LIN {X 0,Y 468.143,Z 375.937,A -85,B 0,C 180,E1 -7618.838,E2 -7618.838} C_VEL
LIN {X 0,Y 467.826,Z 382.891,A -85,B 0,C 180,E1 -7621.757,E2 -7621.757} C_VEL
LIN {X 0,Y 467.602,Z 389.263,A -85,B 0,C 180,E1 -7624.395,E2 -7624.395} C_VEL
LIN {X 0,Y 467.33,Z 397.834,A -85,B 0,C 180,E1 -7627.916,E2 -7627.916} C_VEL
LIN {X 0,Y 467.292,Z 398.559,A -85,B 0,C 180,E1 -7628.21,E2 -7628.21} C_VEL
LIN {X 0,Y 471.188,Z 415.228,A -85,B 0,C 180,E1 -7628.746,E2 -7628.746} C_VEL
LIN {X 0,Y 473.512,Z 427.366,A -85,B 0,C 180,E1 -7629.238,E2 -7629.238} C_VEL
LIN {X 0,Y 472.916,Z 441.368,A -85,B 0,C 180,E1 -7629.804,E2 -7629.804} C_VEL
LIN {X 0,Y 472.102,Z 455.526,A -85,B 0,C 180,E1 -7630.544,E2 -7630.544} C_VEL
LIN {X 0,Y 471.29,Z 468.776,A -85,B 0,C 180,E1 -7631.413,E2 -7631.413} C_VEL
LIN {X 0,Y 470.385,Z 482.274,A -85,B 0,C 180,E1 -7632.502,E2 -7632.502} C_VEL
LIN {X 0,Y 469.612,Z 494.581,A -85,B 0,C 180,E1 -7633.704,E2 -7633.704} C_VEL
LIN {X 0,Y 468.781,Z 505.819,A -85,B 0,C 180,E1 -7635.013,E2 -7635.013} C_VEL
LIN {X 0,Y 468.067,Z 516.736,A -85,B 0,C 180,E1 -7636.542,E2 -7636.542} C_VEL
LIN {X 0,Y 467.596,Z 525.839,A -85,B 0,C 180,E1 -7638.073,E2 -7638.073} C_VEL
LIN {X 0,Y 467.244,Z 533.393,A -85,B 0,C 180,E1 -7639.602,E2 -7639.602} C_VEL
LIN {X 0,Y 466.93,Z 540.444,A -85,B 0,C 180,E1 -7641.344,E2 -7641.344} C_VEL
LIN {X 0,Y 466.818,Z 545.996,A -85,B 0,C 180,E1 -7643.083,E2 -7643.083} C_VEL
LIN {X 0,Y 466.694,Z 550.191,A -85,B 0,C 180,E1 -7644.816,E2 -7644.816} C_VEL
LIN {X 0,Y 466.705,Z 553.137,A -85,B 0,C 180,E1 -7646.547,E2 -7646.547} C_VEL
LIN {X 0,Y 466.652,Z 554.892,A -85,B 0,C 180,E1 -7648.274,E2 -7648.274} C_VEL
LIN {X 0,Y 466.595,Z 555.491,A -85,B 0,C 180,E1 -7650,E2 -7650} C_VEL
LIN {X 0,Y 466.652,Z 554.889,A -85,B 0,C 180,E1 -7651.726,E2 -7651.726} C_VEL
LIN {X 0,Y 466.705,Z 553.132,A -85,B 0,C 180,E1 -7653.454,E2 -7653.454} C_VEL
LIN {X 0,Y 466.721,Z 550.189,A -85,B 0,C 180,E1 -7655.184,E2 -7655.184} C_VEL
LIN {X 0,Y 466.822,Z 545.998,A -85,B 0,C 180,E1 -7656.918,E2 -7656.918} C_VEL
LIN {X 0,Y 466.93,Z 540.443,A -85,B 0,C 180,E1 -7658.657,E2 -7658.657} C_VEL
LIN {X 0,Y 467.245,Z 533.383,A -85,B 0,C 180,E1 -7660.399,E2 -7660.399} C_VEL
LIN {X 0,Y 467.612,Z 525.832,A -85,B 0,C 180,E1 -7661.927,E2 -7661.927} C_VEL
LIN {X 0,Y 468.068,Z 516.733,A -85,B 0,C 180,E1 -7663.458,E2 -7663.458} C_VEL
LIN {X 0,Y 468.76,Z 505.812,A -85,B 0,C 180,E1 -7664.989,E2 -7664.989} C_VEL
LIN {X 0,Y 469.61,Z 493.547,A -85,B 0,C 180,E1 -7666.408,E2 -7666.408} C_VEL
LIN {X 0,Y 470.458,Z 481.048,A -85,B 0,C 180,E1 -7667.609,E2 -7667.609} C_VEL
LIN {X 0,Y 471.366,Z 467.232,A -85,B 0,C 180,E1 -7668.697,E2 -7668.697} C_VEL
LIN {X 0,Y 472.233,Z 453.677,A -85,B 0,C 180,E1 -7669.564,E2 -7669.564} C_VEL
LIN {X 0,Y 472.939,Z 439.651,A -85,B 0,C 180,E1 -7670.28,E2 -7670.28} C_VEL
LIN {X 0,Y 473.403,Z 425.835,A -85,B 0,C 180,E1 -7670.823,E2 -7670.823} C_VEL
LIN {X 0,Y 470.06,Z 410.115,A -85,B 0,C 180,E1 -7671.434,E2 -7671.434} C_VEL
LIN {X 0,Y 467.287,Z 398.544,A -85,B 0,C 180,E1 -7671.794,E2 -7671.794} C_VEL
LIN {X 0,Y 467.513,Z 390.984,A -85,B 0,C 180,E1 -7674.893,E2 -7674.893} C_VEL
LIN {X 0,Y 467.773,Z 384.017,A -85,B 0,C 180,E1 -7677.759,E2 -7677.759} C_VEL
LIN {X 0,Y 468.035,Z 376.994,A -85,B 0,C 180,E1 -7680.7,E2 -7680.7} C_VEL
LIN {X 0,Y 468.345,Z 369.941,A -85,B 0,C 180,E1 -7683.726,E2 -7683.726} C_VEL
LIN {X 0,Y 468.684,Z 364.077,A -85,B 0,C 180,E1 -7686.34,E2 -7686.34} C_VEL
LIN {X 0,Y 468.997,Z 357.229,A -85,B 0,C 180,E1 -7689.559,E2 -7689.559} C_VEL
LIN {X 0,Y 469.127,Z 353.286,A -85,B 0,C 180,E1 -7691.492,E2 -7691.492} C_VEL
LIN {X 0,Y 468.587,Z 348.664,A -85,B 0,C 180,E1 -7693.952,E2 -7693.952} C_VEL
LIN {X 0,Y 467.687,Z 343.617,A -85,B 0,C 180,E1 -7696.865,E2 -7696.865} C_VEL
LIN {X 0,Y 467.591,Z 342.867,A -85,B 0,C 180,E1 -7697.44,E2 -7697.44} C_VEL
LIN {X 0,Y 467.584,Z 342.869,A -85,B 0,C 180,E1 -7700.856,E2 -7700.856} C_VEL
LIN {X 0,Y 467.566,Z 342.872,A -85,B 0,C 180,E1 -7704.261,E2 -7704.261} C_VEL
LIN {X 0,Y 467.584,Z 342.868,A -85,B 0,C 180,E1 -7707.321,E2 -7707.321} C_VEL
LIN {X 0,Y 467.573,Z 342.87,A -85,B 0,C 180,E1 -7710.668,E2 -7710.668} C_VEL
LIN {X 0,Y 467.618,Z 342.862,A -85,B 0,C 180,E1 -7713.2,E2 -7713.2} C_VEL
LIN {X 0,Y 467.595,Z 342.864,A -85,B 0,C 180,E1 -7716.468,E2 -7716.468} C_VEL
LIN {X 0,Y 467.626,Z 342.863,A -85,B 0,C 180,E1 -7719.777,E2 -7719.777} C_VEL
LIN {X 0,Y 467.612,Z 342.862,A -85,B 0,C 180,E1 -7722.507,E2 -7722.507} C_VEL
LIN {X 0,Y 467.61,Z 342.864,A -85,B 0,C 180,E1 -7725.197,E2 -7725.197} C_VEL
LIN {X 0,Y 467.659,Z 342.86,A -85,B 0,C 180,E1 -7727.855,E2 -7727.855} C_VEL
LIN {X 0,Y 467.685,Z 342.853,A -85,B 0,C 180,E1 -7731.357,E2 -7731.357} C_VEL
LIN {X 0,Y 467.747,Z 342.847,A -85,B 0,C 180,E1 -7733.963,E2 -7733.963} C_VEL
LIN {X 0,Y 467.863,Z 342.83,A -85,B 0,C 180,E1 -7737.417,E2 -7737.417} C_VEL
LIN {X 0,Y 467.885,Z 342.829,A -85,B 0,C 180,E1 -7740,E2 -7740} C_VEL
LIN {X 0,Y 467.863,Z 342.832,A -85,B 0,C 180,E1 -7742.583,E2 -7742.583} C_VEL
LIN {X 0,Y 467.748,Z 342.846,A -85,B 0,C 180,E1 -7746.037,E2 -7746.037} C_VEL
LIN {X 0,Y 467.686,Z 342.854,A -85,B 0,C 180,E1 -7748.643,E2 -7748.643} C_VEL
LIN {X 0,Y 467.659,Z 342.844,A -85,B 0,C 180,E1 -7752.145,E2 -7752.145} C_VEL
LIN {X 0,Y 467.643,Z 342.856,A -85,B 0,C 180,E1 -7755.695,E2 -7755.695} C_VEL
LIN {X 0,Y 467.621,Z 342.855,A -85,B 0,C 180,E1 -7758.765,E2 -7758.765} C_VEL
LIN {X 0,Y 467.584,Z 342.858,A -85,B 0,C 180,E1 -7761.268,E2 -7761.268} C_VEL
LIN {X 0,Y 467.566,Z 342.869,A -85,B 0,C 180,E1 -7763.944,E2 -7763.944} C_VEL
LIN {X 0,Y 467.616,Z 342.855,A -85,B 0,C 180,E1 -7766.8,E2 -7766.8} C_VEL
LIN {X 0,Y 467.557,Z 342.868,A -85,B 0,C 180,E1 -7769.738,E2 -7769.738} C_VEL
LIN {X 0,Y 467.586,Z 342.86,A -85,B 0,C 180,E1 -7772.758,E2 -7772.758} C_VEL
LIN {X 0,Y 467.559,Z 342.868,A -85,B 0,C 180,E1 -7775.889,E2 -7775.889} C_VEL
LIN {X 0,Y 467.586,Z 342.867,A -85,B 0,C 180,E1 -7779.145,E2 -7779.145} C_VEL
LIN {X 0,Y 467.589,Z 342.869,A -85,B 0,C 180,E1 -7782.567,E2 -7782.567} C_VEL
LIN {X 0,Y 467.573,Z 342.869,A -85,B 0,C 180,E1 -7785.053,E2 -7785.053} C_VEL
LIN {X 0,Y 467.545,Z 342.874,A -85,B 0,C 180,E1 -7787.439,E2 -7787.439} C_VEL
LIN {X 0,Y 467.333,Z 342.9,A -85,B 0,C 180,E1 -7790.082,E2 -7790.082} C_VEL
LIN {X 0,Y 467.23,Z 343.077,A -85,B 0,C 180,E1 -7791.46,E2 -7791.46} C_VEL
LIN {X 0,Y 467.185,Z 345.526,A -85,B 0,C 180,E1 -7794.325,E2 -7794.325} C_VEL
LIN {X 0,Y 467.138,Z 348.226,A -85,B 0,C 180,E1 -7797.406,E2 -7797.406} C_VEL
LIN {X 0,Y 467.036,Z 351.246,A -85,B 0,C 180,E1 -7800.785,E2 -7800.785} C_VEL
LIN {X 0,Y 466.95,Z 354.424,A -85,B 0,C 180,E1 -7804.12,E2 -7804.12} C_VEL
LIN {X 0,Y 466.89,Z 357.26,A -85,B 0,C 180,E1 -7806.96,E2 -7806.96} C_VEL
LIN {X 0,Y 466.856,Z 358.631,A -85,B 0,C 180,E1 -7808.273,E2 -7808.273} C_VEL
LIN {X 0,Y 472.012,Z 374.868,A -85,B 0,C 180,E1 -7808.908,E2 -7808.908} C_VEL
LIN {X 0,Y 473.883,Z 382.02,A -85,B 0,C 180,E1 -7809.228,E2 -7809.228} C_VEL
LIN {X 0,Y 473.379,Z 397.457,A -85,B 0,C 180,E1 -7809.851,E2 -7809.851} C_VEL
LIN {X 0,Y 472.672,Z 411.134,A -85,B 0,C 180,E1 -7810.568,E2 -7810.568} C_VEL
LIN {X 0,Y 472.562,Z 413.419,A -85,B 0,C 180,E1 -7810.71,E2 -7810.71} C_VEL
LIN {X 0,Y 471.674,Z 418.718,A -85,B 0,C 180,E1 -7811.02,E2 -7811.02} C_VEL
LIN {X 0,Y 468.437,Z 427.17,A -85,B 0,C 180,E1 -7811.503,E2 -7811.503} C_VEL
LIN {X 0,Y 465.109,Z 435.383,A -85,B 0,C 180,E1 -7812.047,E2 -7812.047} C_VEL
LIN {X 0,Y 464.087,Z 440.168,A -85,B 0,C 180,E1 -7812.453,E2 -7812.453} C_VEL
LIN {X 0,Y 463.172,Z 452.261,A -85,B 0,C 180,E1 -7813.697,E2 -7813.697} C_VEL
LIN {X 0,Y 462.349,Z 463.033,A -85,B 0,C 180,E1 -7815.024,E2 -7815.024} C_VEL
LIN {X 0,Y 461.661,Z 472.162,A -85,B 0,C 180,E1 -7816.351,E2 -7816.351} C_VEL
LIN {X 0,Y 461.067,Z 481.078,A -85,B 0,C 180,E1 -7817.901,E2 -7817.901} C_VEL
LIN {X 0,Y 460.524,Z 488.466,A -85,B 0,C 180,E1 -7819.447,E2 -7819.447} C_VEL
LIN {X 0,Y 460.187,Z 495.365,A -85,B 0,C 180,E1 -7821.215,E2 -7821.215} C_VEL
LIN {X 0,Y 459.916,Z 500.786,A -85,B 0,C 180,E1 -7822.978,E2 -7822.978} C_VEL
LIN {X 0,Y 459.699,Z 504.881,A -85,B 0,C 180,E1 -7824.737,E2 -7824.737} C_VEL
LIN {X 0,Y 459.689,Z 507.753,A -85,B 0,C 180,E1 -7826.494,E2 -7826.494} C_VEL
LIN {X 0,Y 459.631,Z 509.485,A -85,B 0,C 180,E1 -7828.247,E2 -7828.247} C_VEL
LIN {X 0,Y 459.528,Z 510.096,A -85,B 0,C 180,E1 -7830,E2 -7830} C_VEL
LIN {X 0,Y 459.632,Z 509.536,A -85,B 0,C 180,E1 -7831.752,E2 -7831.752} C_VEL
LIN {X 0,Y 459.689,Z 507.872,A -85,B 0,C 180,E1 -7833.506,E2 -7833.506} C_VEL
LIN {X 0,Y 459.694,Z 505.065,A -85,B 0,C 180,E1 -7835.263,E2 -7835.263} C_VEL
LIN {X 0,Y 459.908,Z 501.035,A -85,B 0,C 180,E1 -7837.022,E2 -7837.022} C_VEL
LIN {X 0,Y 460.182,Z 495.691,A -85,B 0,C 180,E1 -7838.784,E2 -7838.784} C_VEL
LIN {X 0,Y 460.498,Z 488.881,A -85,B 0,C 180,E1 -7840.552,E2 -7840.552} C_VEL
LIN {X 0,Y 461.022,Z 481.546,A -85,B 0,C 180,E1 -7842.099,E2 -7842.099} C_VEL
LIN {X 0,Y 461.624,Z 472.707,A -85,B 0,C 180,E1 -7843.649,E2 -7843.649} C_VEL
LIN {X 0,Y 462.296,Z 463.688,A -85,B 0,C 180,E1 -7844.977,E2 -7844.977} C_VEL
LIN {X 0,Y 463.089,Z 453.042,A -85,B 0,C 180,E1 -7846.305,E2 -7846.305} C_VEL
LIN {X 0,Y 463.997,Z 441.752,A -85,B 0,C 180,E1 -7847.486,E2 -7847.486} C_VEL
LIN {X 0,Y 464.916,Z 428.697,A -85,B 0,C 180,E1 -7848.623,E2 -7848.623} C_VEL
LIN {X 0,Y 465.751,Z 414.664,A -85,B 0,C 180,E1 -7849.617,E2 -7849.617} C_VEL
LIN {X 0,Y 466.589,Z 400.159,A -85,B 0,C 180,E1 -7850.427,E2 -7850.427} C_VEL
LIN {X 0,Y 467.191,Z 384.917,A -85,B 0,C 180,E1 -7851.078,E2 -7851.078} C_VEL
LIN {X 0,Y 467.053,Z 382.296,A -85,B 0,C 180,E1 -7851.184,E2 -7851.184} C_VEL
LIN {X 0,Y 462.919,Z 368.608,A -85,B 0,C 180,E1 -7851.802,E2 -7851.802} C_VEL
LIN {X 0,Y 459.771,Z 358.928,A -85,B 0,C 180,E1 -7852.186,E2 -7852.186} C_VEL
LIN {X 0,Y 459.889,Z 355.488,A -85,B 0,C 180,E1 -7855.626,E2 -7855.626} C_VEL
LIN {X 0,Y 459.941,Z 352.956,A -85,B 0,C 180,E1 -7858.273,E2 -7858.273} C_VEL
LIN {X 0,Y 460.006,Z 350.233,A -85,B 0,C 180,E1 -7861.295,E2 -7861.295} C_VEL
LIN {X 0,Y 460.124,Z 347.516,A -85,B 0,C 180,E1 -7864.431,E2 -7864.431} C_VEL
LIN {X 0,Y 460.157,Z 344.726,A -85,B 0,C 180,E1 -7867.656,E2 -7867.656} C_VEL
LIN {X 0,Y 460.17,Z 343.794,A -85,B 0,C 180,E1 -7868.84,E2 -7868.84} C_VEL
LIN {X 0,Y 460.455,Z 343.754,A -85,B 0,C 180,E1 -7871.591,E2 -7871.591} C_VEL
LIN {X 0,Y 460.515,Z 343.749,A -85,B 0,C 180,E1 -7874.588,E2 -7874.588} C_VEL
LIN {X 0,Y 460.521,Z 343.748,A -85,B 0,C 180,E1 -7877.818,E2 -7877.818} C_VEL
LIN {X 0,Y 460.544,Z 343.742,A -85,B 0,C 180,E1 -7881.102,E2 -7881.102} C_VEL
LIN {X 0,Y 460.513,Z 343.746,A -85,B 0,C 180,E1 -7884.554,E2 -7884.554} C_VEL
LIN {X 0,Y 460.531,Z 343.738,A -85,B 0,C 180,E1 -7887.715,E2 -7887.715} C_VEL
LIN {X 0,Y 460.546,Z 343.741,A -85,B 0,C 180,E1 -7890.769,E2 -7890.769} C_VEL
LIN {X 0,Y 460.567,Z 343.732,A -85,B 0,C 180,E1 -7893.735,E2 -7893.735} C_VEL
LIN {X 0,Y 460.544,Z 343.741,A -85,B 0,C 180,E1 -7896.624,E2 -7896.624} C_VEL
LIN {X 0,Y 460.55,Z 343.729,A -85,B 0,C 180,E1 -7899.453,E2 -7899.453} C_VEL
LIN {X 0,Y 460.558,Z 343.742,A -85,B 0,C 180,E1 -7902.23,E2 -7902.23} C_VEL
LIN {X 0,Y 460.564,Z 343.738,A -85,B 0,C 180,E1 -7904.965,E2 -7904.965} C_VEL
LIN {X 0,Y 460.628,Z 343.721,A -85,B 0,C 180,E1 -7907.666,E2 -7907.666} C_VEL
LIN {X 0,Y 460.627,Z 343.734,A -85,B 0,C 180,E1 -7911.224,E2 -7911.224} C_VEL
LIN {X 0,Y 460.709,Z 343.723,A -85,B 0,C 180,E1 -7913.87,E2 -7913.87} C_VEL
LIN {X 0,Y 460.823,Z 343.71,A -85,B 0,C 180,E1 -7917.378,E2 -7917.378} C_VEL
LIN {X 0,Y 460.851,Z 343.707,A -85,B 0,C 180,E1 -7920,E2 -7920} C_VEL
LIN {X 0,Y 460.824,Z 343.707,A -85,B 0,C 180,E1 -7922.622,E2 -7922.622} C_VEL
LIN {X 0,Y 460.708,Z 343.725,A -85,B 0,C 180,E1 -7926.13,E2 -7926.13} C_VEL
LIN {X 0,Y 460.627,Z 343.732,A -85,B 0,C 180,E1 -7928.776,E2 -7928.776} C_VEL
LIN {X 0,Y 460.611,Z 343.734,A -85,B 0,C 180,E1 -7932.445,E2 -7932.445} C_VEL
LIN {X 0,Y 460.597,Z 343.734,A -85,B 0,C 180,E1 -7935.998,E2 -7935.998} C_VEL
LIN {X 0,Y 460.569,Z 343.74,A -85,B 0,C 180,E1 -7938.902,E2 -7938.902} C_VEL
LIN {X 0,Y 460.514,Z 343.749,A -85,B 0,C 180,E1 -7941.486,E2 -7941.486} C_VEL
LIN {X 0,Y 460.54,Z 343.746,A -85,B 0,C 180,E1 -7944.332,E2 -7944.332} C_VEL
LIN {X 0,Y 460.577,Z 343.741,A -85,B 0,C 180,E1 -7947.243,E2 -7947.243} C_VEL
LIN {X 0,Y 460.525,Z 343.746,A -85,B 0,C 180,E1 -7950.239,E2 -7950.239} C_VEL
LIN {X 0,Y 460.527,Z 343.747,A -85,B 0,C 180,E1 -7953.325,E2 -7953.325} C_VEL
LIN {X 0,Y 460.477,Z 343.753,A -85,B 0,C 180,E1 -7956.529,E2 -7956.529} C_VEL
LIN {X 0,Y 460.556,Z 343.744,A -85,B 0,C 180,E1 -7959.86,E2 -7959.86} C_VEL
LIN {X 0,Y 460.549,Z 343.823,A -85,B 0,C 180,E1 -7962.368,E2 -7962.368} C_VEL
LIN {X 0,Y 461.49,Z 349.212,A -85,B 0,C 180,E1 -7965.531,E2 -7965.531} C_VEL
LIN {X 0,Y 462.108,Z 354.056,A -85,B 0,C 180,E1 -7968.178,E2 -7968.178} C_VEL
LIN {X 0,Y 462.055,Z 358.224,A -85,B 0,C 180,E1 -7970.296,E2 -7970.296} C_VEL
LIN {X 0,Y 461.674,Z 365.567,A -85,B 0,C 180,E1 -7973.785,E2 -7973.785} C_VEL
LIN {X 0,Y 461.28,Z 372.537,A -85,B 0,C 180,E1 -7976.927,E2 -7976.927} C_VEL
LIN {X 0,Y 460.999,Z 379.111,A -85,B 0,C 180,E1 -7979.796,E2 -7979.796} C_VEL
LIN {X 0,Y 460.668,Z 386.088,A -85,B 0,C 180,E1 -7982.763,E2 -7982.763} C_VEL
LIN {X 0,Y 460.411,Z 392.987,A -85,B 0,C 180,E1 -7985.661,E2 -7985.661} C_VEL
LIN {X 0,Y 460.252,Z 398.18,A -85,B 0,C 180,E1 -7987.848,E2 -7987.848} C_VEL
LIN {X 0,Y 464.531,Z 416.477,A -85,B 0,C 180,E1 -7988.469,E2 -7988.469} C_VEL
LIN {X 0,Y 466.803,Z 428.417,A -85,B 0,C 180,E1 -7988.979,E2 -7988.979} C_VEL
LIN {X 0,Y 466.202,Z 441.436,A -85,B 0,C 180,E1 -7989.521,E2 -7989.521} C_VEL
LIN {X 0,Y 465.391,Z 455.18,A -85,B 0,C 180,E1 -7990.252,E2 -7990.252} C_VEL
LIN {X 0,Y 464.469,Z 468.425,A -85,B 0,C 180,E1 -7991.13,E2 -7991.13} C_VEL
LIN {X 0,Y 463.542,Z 481.925,A -85,B 0,C 180,E1 -7992.235,E2 -7992.235} C_VEL
LIN {X 0,Y 462.707,Z 494.23,A -85,B 0,C 180,E1 -7993.454,E2 -7993.454} C_VEL
LIN {X 0,Y 461.839,Z 505.468,A -85,B 0,C 180,E1 -7994.782,E2 -7994.782} C_VEL
LIN {X 0,Y 461.082,Z 516.385,A -85,B 0,C 180,E1 -7996.335,E2 -7996.335} C_VEL
LIN {X 0,Y 460.551,Z 525.486,A -85,B 0,C 180,E1 -7997.888,E2 -7997.888} C_VEL
LIN {X 0,Y 460.194,Z 533.042,A -85,B 0,C 180,E1 -7999.441,E2 -7999.441} C_VEL
LIN {X 0,Y 459.868,Z 540.094,A -85,B 0,C 180,E1 -8001.21,E2 -8001.21} C_VEL
LIN {X 0,Y 459.728,Z 545.646,A -85,B 0,C 180,E1 -8002.976,E2 -8002.976} C_VEL
LIN {X 0,Y 459.605,Z 549.843,A -85,B 0,C 180,E1 -8004.736,E2 -8004.736} C_VEL
LIN {X 0,Y 459.601,Z 552.789,A -85,B 0,C 180,E1 -8006.494,E2 -8006.494} C_VEL
LIN {X 0,Y 459.56,Z 554.544,A -85,B 0,C 180,E1 -8008.248,E2 -8008.248} C_VEL
LIN {X 0,Y 459.527,Z 555.144,A -85,B 0,C 180,E1 -8010,E2 -8010} C_VEL
LIN {X 0,Y 459.56,Z 554.541,A -85,B 0,C 180,E1 -8011.753,E2 -8011.753} C_VEL
LIN {X 0,Y 459.601,Z 552.783,A -85,B 0,C 180,E1 -8013.507,E2 -8013.507} C_VEL
LIN {X 0,Y 459.631,Z 549.84,A -85,B 0,C 180,E1 -8015.264,E2 -8015.264} C_VEL
LIN {X 0,Y 459.73,Z 545.648,A -85,B 0,C 180,E1 -8017.025,E2 -8017.025} C_VEL
LIN {X 0,Y 459.869,Z 540.093,A -85,B 0,C 180,E1 -8018.791,E2 -8018.791} C_VEL
LIN {X 0,Y 460.195,Z 533.032,A -85,B 0,C 180,E1 -8020.56,E2 -8020.56} C_VEL
LIN {X 0,Y 460.562,Z 525.478,A -85,B 0,C 180,E1 -8022.112,E2 -8022.112} C_VEL
LIN {X 0,Y 461.084,Z 516.38,A -85,B 0,C 180,E1 -8023.666,E2 -8023.666} C_VEL
LIN {X 0,Y 461.812,Z 505.458,A -85,B 0,C 180,E1 -8025.22,E2 -8025.22} C_VEL
LIN {X 0,Y 462.717,Z 493.193,A -85,B 0,C 180,E1 -8026.66,E2 -8026.66} C_VEL
LIN {X 0,Y 463.613,Z 480.694,A -85,B 0,C 180,E1 -8027.877,E2 -8027.877} C_VEL
LIN {X 0,Y 464.603,Z 466.879,A -85,B 0,C 180,E1 -8028.98,E2 -8028.98} C_VEL
LIN {X 0,Y 465.519,Z 453.324,A -85,B 0,C 180,E1 -8029.858,E2 -8029.858} C_VEL
LIN {X 0,Y 466.252,Z 438.42,A -85,B 0,C 180,E1 -8030.625,E2 -8030.625} C_VEL
LIN {X 0,Y 466.736,Z 427.317,A -85,B 0,C 180,E1 -8031.066,E2 -8031.066} C_VEL
LIN {X 0,Y 463.453,Z 411.48,A -85,B 0,C 180,E1 -8031.711,E2 -8031.711} C_VEL
LIN {X 0,Y 460.254,Z 398.191,A -85,B 0,C 180,E1 -8032.145,E2 -8032.145} C_VEL
LIN {X 0,Y 460.581,Z 389.454,A -85,B 0,C 180,E1 -8035.805,E2 -8035.805} C_VEL
LIN {X 0,Y 460.894,Z 381.437,A -85,B 0,C 180,E1 -8039.207,E2 -8039.207} C_VEL
LIN {X 0,Y 461.193,Z 374.372,A -85,B 0,C 180,E1 -8042.233,E2 -8042.233} C_VEL
LIN {X 0,Y 461.538,Z 367.371,A -85,B 0,C 180,E1 -8045.355,E2 -8045.355} C_VEL
LIN {X 0,Y 461.776,Z 362.393,A -85,B 0,C 180,E1 -8047.682,E2 -8047.682} C_VEL
LIN {X 0,Y 462.141,Z 355.905,A -85,B 0,C 180,E1 -8050.838,E2 -8050.838} C_VEL
LIN {X 0,Y 461.835,Z 351.65,A -85,B 0,C 180,E1 -8053.077,E2 -8053.077} C_VEL
LIN {X 0,Y 461.091,Z 346.925,A -85,B 0,C 180,E1 -8055.757,E2 -8055.757} C_VEL
LIN {X 0,Y 460.526,Z 343.748,A -85,B 0,C 180,E1 -8057.724,E2 -8057.724} C_VEL
LIN {X 0,Y 460.547,Z 343.746,A -85,B 0,C 180,E1 -8061.103,E2 -8061.103} C_VEL
LIN {X 0,Y 460.516,Z 343.75,A -85,B 0,C 180,E1 -8064.555,E2 -8064.555} C_VEL
LIN {X 0,Y 460.534,Z 343.746,A -85,B 0,C 180,E1 -8067.716,E2 -8067.716} C_VEL
LIN {X 0,Y 460.543,Z 343.746,A -85,B 0,C 180,E1 -8070.769,E2 -8070.769} C_VEL
LIN {X 0,Y 460.562,Z 343.743,A -85,B 0,C 180,E1 -8073.735,E2 -8073.735} C_VEL
LIN {X 0,Y 460.548,Z 343.743,A -85,B 0,C 180,E1 -8076.624,E2 -8076.624} C_VEL
LIN {X 0,Y 460.554,Z 343.741,A -85,B 0,C 180,E1 -8079.453,E2 -8079.453} C_VEL
LIN {X 0,Y 460.562,Z 343.74,A -85,B 0,C 180,E1 -8082.23,E2 -8082.23} C_VEL
LIN {X 0,Y 460.569,Z 343.742,A -85,B 0,C 180,E1 -8084.965,E2 -8084.965} C_VEL
LIN {X 0,Y 460.614,Z 343.735,A -85,B 0,C 180,E1 -8088.559,E2 -8088.559} C_VEL
LIN {X 0,Y 460.699,Z 343.728,A -85,B 0,C 180,E1 -8092.109,E2 -8092.109} C_VEL
LIN {X 0,Y 460.7,Z 343.723,A -85,B 0,C 180,E1 -8094.748,E2 -8094.748} C_VEL
LIN {X 0,Y 460.828,Z 343.706,A -85,B 0,C 180,E1 -8097.378,E2 -8097.378} C_VEL
LIN {X 0,Y 460.856,Z 343.705,A -85,B 0,C 180,E1 -8100,E2 -8100} C_VEL
LIN {X 0,Y 460.827,Z 343.709,A -85,B 0,C 180,E1 -8102.622,E2 -8102.622} C_VEL
LIN {X 0,Y 460.714,Z 343.721,A -85,B 0,C 180,E1 -8106.13,E2 -8106.13} C_VEL
LIN {X 0,Y 460.633,Z 343.734,A -85,B 0,C 180,E1 -8108.776,E2 -8108.776} C_VEL
LIN {X 0,Y 460.617,Z 343.718,A -85,B 0,C 180,E1 -8112.445,E2 -8112.445} C_VEL
LIN {X 0,Y 460.604,Z 343.733,A -85,B 0,C 180,E1 -8115.998,E2 -8115.998} C_VEL
LIN {X 0,Y 460.574,Z 343.733,A -85,B 0,C 180,E1 -8118.902,E2 -8118.902} C_VEL
LIN {X 0,Y 460.519,Z 343.741,A -85,B 0,C 180,E1 -8121.486,E2 -8121.486} C_VEL
LIN {X 0,Y 460.534,Z 343.745,A -85,B 0,C 180,E1 -8124.333,E2 -8124.333} C_VEL
LIN {X 0,Y 460.574,Z 343.73,A -85,B 0,C 180,E1 -8127.244,E2 -8127.244} C_VEL
LIN {X 0,Y 460.514,Z 343.749,A -85,B 0,C 180,E1 -8130.24,E2 -8130.24} C_VEL
LIN {X 0,Y 460.532,Z 343.738,A -85,B 0,C 180,E1 -8133.325,E2 -8133.325} C_VEL
LIN {X 0,Y 460.482,Z 343.753,A -85,B 0,C 180,E1 -8136.529,E2 -8136.529} C_VEL
LIN {X 0,Y 460.561,Z 343.741,A -85,B 0,C 180,E1 -8139.859,E2 -8139.859} C_VEL
LIN {X 0,Y 460.516,Z 343.748,A -85,B 0,C 180,E1 -8142.9,E2 -8142.9} C_VEL
LIN {X 0,Y 460.513,Z 343.75,A -85,B 0,C 180,E1 -8145.83,E2 -8145.83} C_VEL
LIN {X 0,Y 460.398,Z 343.766,A -85,B 0,C 180,E1 -8148.974,E2 -8148.974} C_VEL
LIN {X 0,Y 460.179,Z 343.792,A -85,B 0,C 180,E1 -8151.232,E2 -8151.232} C_VEL
LIN {X 0,Y 460.122,Z 346.495,A -85,B 0,C 180,E1 -8154.52,E2 -8154.52} C_VEL
LIN {X 0,Y 460.054,Z 349.225,A -85,B 0,C 180,E1 -8157.678,E2 -8157.678} C_VEL
LIN {X 0,Y 459.999,Z 351.927,A -85,B 0,C 180,E1 -8160.731,E2 -8160.731} C_VEL
LIN {X 0,Y 459.882,Z 354.733,A -85,B 0,C 180,E1 -8163.692,E2 -8163.692} C_VEL
LIN {X 0,Y 459.813,Z 357.593,A -85,B 0,C 180,E1 -8166.584,E2 -8166.584} C_VEL
LIN {X 0,Y 459.8,Z 359.129,A -85,B 0,C 180,E1 -8167.929,E2 -8167.929} C_VEL
LIN {X 0,Y 464.762,Z 374.228,A -85,B 0,C 180,E1 -8168.53,E2 -8168.53} C_VEL
LIN {X 0,Y 467.208,Z 383.219,A -85,B 0,C 180,E1 -8168.949,E2 -8168.949} C_VEL
LIN {X 0,Y 466.733,Z 398.085,A -85,B 0,C 180,E1 -8169.565,E2 -8169.565} C_VEL
LIN {X 0,Y 465.979,Z 411.489,A -85,B 0,C 180,E1 -8170.277,E2 -8170.277} C_VEL
LIN {X 0,Y 465.215,Z 424.713,A -85,B 0,C 180,E1 -8171.161,E2 -8171.161} C_VEL
LIN {X 0,Y 464.261,Z 438.148,A -85,B 0,C 180,E1 -8172.262,E2 -8172.262} C_VEL
LIN {X 0,Y 464.087,Z 440.168,A -85,B 0,C 180,E1 -8172.453,E2 -8172.453} C_VEL
LIN {X 0,Y 463.067,Z 444.902,A -85,B 0,C 180,E1 -8172.88,E2 -8172.88} C_VEL
LIN {X 0,Y 459.687,Z 452.416,A -85,B 0,C 180,E1 -8173.566,E2 -8173.566} C_VEL
LIN {X 0,Y 456.373,Z 459.592,A -85,B 0,C 180,E1 -8174.312,E2 -8174.312} C_VEL
LIN {X 0,Y 455.448,Z 463.679,A -85,B 0,C 180,E1 -8174.833,E2 -8174.833} C_VEL
LIN {X 0,Y 454.631,Z 473.852,A -85,B 0,C 180,E1 -8176.364,E2 -8176.364} C_VEL
LIN {X 0,Y 454.06,Z 482.541,A -85,B 0,C 180,E1 -8177.939,E2 -8177.939} C_VEL
LIN {X 0,Y 453.522,Z 488.818,A -85,B 0,C 180,E1 -8179.283,E2 -8179.283} C_VEL
LIN {X 0,Y 453.142,Z 495.716,A -85,B 0,C 180,E1 -8181.077,E2 -8181.077} C_VEL
LIN {X 0,Y 452.857,Z 501.136,A -85,B 0,C 180,E1 -8182.868,E2 -8182.868} C_VEL
LIN {X 0,Y 452.643,Z 505.229,A -85,B 0,C 180,E1 -8184.654,E2 -8184.654} C_VEL
LIN {X 0,Y 452.624,Z 508.1,A -85,B 0,C 180,E1 -8186.439,E2 -8186.439} C_VEL
LIN {X 0,Y 452.541,Z 509.833,A -85,B 0,C 180,E1 -8188.22,E2 -8188.22} C_VEL
LIN {X 0,Y 452.462,Z 510.442,A -85,B 0,C 180,E1 -8190,E2 -8190} C_VEL
LIN {X 0,Y 452.541,Z 509.884,A -85,B 0,C 180,E1 -8191.78,E2 -8191.78} C_VEL
LIN {X 0,Y 452.624,Z 508.219,A -85,B 0,C 180,E1 -8193.56,E2 -8193.56} C_VEL
LIN {X 0,Y 452.638,Z 505.411,A -85,B 0,C 180,E1 -8195.345,E2 -8195.345} C_VEL
LIN {X 0,Y 452.852,Z 501.382,A -85,B 0,C 180,E1 -8197.132,E2 -8197.132} C_VEL
LIN {X 0,Y 453.135,Z 496.038,A -85,B 0,C 180,E1 -8198.922,E2 -8198.922} C_VEL
LIN {X 0,Y 453.498,Z 489.228,A -85,B 0,C 180,E1 -8200.717,E2 -8200.717} C_VEL
LIN {X 0,Y 454.065,Z 481.892,A -85,B 0,C 180,E1 -8202.287,E2 -8202.287} C_VEL
LIN {X 0,Y 454.703,Z 473.054,A -85,B 0,C 180,E1 -8203.861,E2 -8203.861} C_VEL
LIN {X 0,Y 455.42,Z 464.034,A -85,B 0,C 180,E1 -8205.209,E2 -8205.209} C_VEL
LIN {X 0,Y 456.256,Z 453.387,A -85,B 0,C 180,E1 -8206.556,E2 -8206.556} C_VEL
LIN {X 0,Y 457.211,Z 442.325,A -85,B 0,C 180,E1 -8207.731,E2 -8207.731} C_VEL
LIN {X 0,Y 458.077,Z 430.455,A -85,B 0,C 180,E1 -8208.795,E2 -8208.795} C_VEL
LIN {X 0,Y 458.924,Z 418.477,A -85,B 0,C 180,E1 -8209.688,E2 -8209.688} C_VEL
LIN {X 0,Y 459.73,Z 404.61,A -85,B 0,C 180,E1 -8210.527,E2 -8210.527} C_VEL
LIN {X 0,Y 460.416,Z 389.888,A -85,B 0,C 180,E1 -8211.219,E2 -8211.219} C_VEL
LIN {X 0,Y 460.473,Z 384.003,A -85,B 0,C 180,E1 -8211.449,E2 -8211.449} C_VEL
LIN {X 0,Y 456.087,Z 369.464,A -85,B 0,C 180,E1 -8212.132,E2 -8212.132} C_VEL
LIN {X 0,Y 452.798,Z 359.861,A -85,B 0,C 180,E1 -8212.516,E2 -8212.516} C_VEL
LIN {X 0,Y 452.739,Z 359.286,A -85,B 0,C 180,E1 -8212.533,E2 -8212.533} C_VEL
LIN {X 0,Y 452.818,Z 356.034,A -85,B 0,C 180,E1 -8215.816,E2 -8215.816} C_VEL
LIN {X 0,Y 452.9,Z 353.254,A -85,B 0,C 180,E1 -8218.754,E2 -8218.754} C_VEL
LIN {X 0,Y 452.956,Z 350.505,A -85,B 0,C 180,E1 -8221.839,E2 -8221.839} C_VEL
LIN {X 0,Y 453.066,Z 347.789,A -85,B 0,C 180,E1 -8225.025,E2 -8225.025} C_VEL
LIN {X 0,Y 453.118,Z 344.939,A -85,B 0,C 180,E1 -8228.346,E2 -8228.346} C_VEL
LIN {X 0,Y 453.321,Z 344.643,A -85,B 0,C 180,E1 -8230.627,E2 -8230.627} C_VEL
LIN {X 0,Y 453.477,Z 344.623,A -85,B 0,C 180,E1 -8233.247,E2 -8233.247} C_VEL
LIN {X 0,Y 453.465,Z 344.625,A -85,B 0,C 180,E1 -8235.779,E2 -8235.779} C_VEL
LIN {X 0,Y 453.478,Z 344.623,A -85,B 0,C 180,E1 -8238.209,E2 -8238.209} C_VEL
LIN {X 0,Y 453.514,Z 344.62,A -85,B 0,C 180,E1 -8240.79,E2 -8240.79} C_VEL
LIN {X 0,Y 453.456,Z 344.628,A -85,B 0,C 180,E1 -8243.917,E2 -8243.917} C_VEL
LIN {X 0,Y 453.481,Z 344.616,A -85,B 0,C 180,E1 -8247.151,E2 -8247.151} C_VEL
LIN {X 0,Y 453.512,Z 344.618,A -85,B 0,C 180,E1 -8250.271,E2 -8250.271} C_VEL
LIN {X 0,Y 453.512,Z 344.611,A -85,B 0,C 180,E1 -8253.294,E2 -8253.294} C_VEL
LIN {X 0,Y 453.502,Z 344.62,A -85,B 0,C 180,E1 -8256.239,E2 -8256.239} C_VEL
LIN {X 0,Y 453.481,Z 344.611,A -85,B 0,C 180,E1 -8259.117,E2 -8259.117} C_VEL
LIN {X 0,Y 453.511,Z 344.618,A -85,B 0,C 180,E1 -8261.944,E2 -8261.944} C_VEL
LIN {X 0,Y 453.538,Z 344.615,A -85,B 0,C 180,E1 -8264.726,E2 -8264.726} C_VEL
LIN {X 0,Y 453.6,Z 344.595,A -85,B 0,C 180,E1 -8267.472,E2 -8267.472} C_VEL
LIN {X 0,Y 453.591,Z 344.612,A -85,B 0,C 180,E1 -8271.087,E2 -8271.087} C_VEL
LIN {X 0,Y 453.676,Z 344.599,A -85,B 0,C 180,E1 -8273.775,E2 -8273.775} C_VEL
LIN {X 0,Y 453.764,Z 344.59,A -85,B 0,C 180,E1 -8277.337,E2 -8277.337} C_VEL
LIN {X 0,Y 453.822,Z 344.582,A -85,B 0,C 180,E1 -8280,E2 -8280} C_VEL
LIN {X 0,Y 453.764,Z 344.586,A -85,B 0,C 180,E1 -8282.663,E2 -8282.663} C_VEL
LIN {X 0,Y 453.676,Z 344.602,A -85,B 0,C 180,E1 -8286.225,E2 -8286.225} C_VEL
LIN {X 0,Y 453.591,Z 344.609,A -85,B 0,C 180,E1 -8288.913,E2 -8288.913} C_VEL
LIN {X 0,Y 453.561,Z 344.612,A -85,B 0,C 180,E1 -8292.529,E2 -8292.529} C_VEL
LIN {X 0,Y 453.542,Z 344.613,A -85,B 0,C 180,E1 -8296.196,E2 -8296.196} C_VEL
LIN {X 0,Y 453.518,Z 344.618,A -85,B 0,C 180,E1 -8299.041,E2 -8299.041} C_VEL
LIN {X 0,Y 453.474,Z 344.625,A -85,B 0,C 180,E1 -8301.836,E2 -8301.836} C_VEL
LIN {X 0,Y 453.512,Z 344.622,A -85,B 0,C 180,E1 -8304.734,E2 -8304.734} C_VEL
LIN {X 0,Y 453.536,Z 344.618,A -85,B 0,C 180,E1 -8307.961,E2 -8307.961} C_VEL
LIN {X 0,Y 453.481,Z 344.626,A -85,B 0,C 180,E1 -8310.759,E2 -8310.759} C_VEL
LIN {X 0,Y 453.476,Z 344.625,A -85,B 0,C 180,E1 -8313.913,E2 -8313.913} C_VEL
LIN {X 0,Y 453.468,Z 344.626,A -85,B 0,C 180,E1 -8317.188,E2 -8317.188} C_VEL
LIN {X 0,Y 453.515,Z 344.62,A -85,B 0,C 180,E1 -8319.447,E2 -8319.447} C_VEL
LIN {X 0,Y 453.503,Z 344.716,A -85,B 0,C 180,E1 -8322,E2 -8322} C_VEL
LIN {X 0,Y 454.27,Z 348.997,A -85,B 0,C 180,E1 -8324.63,E2 -8324.63} C_VEL
LIN {X 0,Y 455.094,Z 354.728,A -85,B 0,C 180,E1 -8327.839,E2 -8327.839} C_VEL
LIN {X 0,Y 455.161,Z 358.04,A -85,B 0,C 180,E1 -8329.571,E2 -8329.571} C_VEL
LIN {X 0,Y 454.734,Z 364.917,A -85,B 0,C 180,E1 -8332.933,E2 -8332.933} C_VEL
LIN {X 0,Y 454.346,Z 371.872,A -85,B 0,C 180,E1 -8336.161,E2 -8336.161} C_VEL
LIN {X 0,Y 454.023,Z 378.841,A -85,B 0,C 180,E1 -8339.282,E2 -8339.282} C_VEL
LIN {X 0,Y 453.665,Z 385.796,A -85,B 0,C 180,E1 -8342.307,E2 -8342.307} C_VEL
LIN {X 0,Y 453.381,Z 392.668,A -85,B 0,C 180,E1 -8345.258,E2 -8345.258} C_VEL
LIN {X 0,Y 453.222,Z 397.839,A -85,B 0,C 180,E1 -8347.482,E2 -8347.482} C_VEL
LIN {X 0,Y 457.655,Z 416.574,A -85,B 0,C 180,E1 -8348.143,E2 -8348.143} C_VEL
LIN {X 0,Y 460.07,Z 429.378,A -85,B 0,C 180,E1 -8348.706,E2 -8348.706} C_VEL
LIN {X 0,Y 459.409,Z 443.202,A -85,B 0,C 180,E1 -8349.313,E2 -8349.313} C_VEL
LIN {X 0,Y 458.545,Z 456.608,A -85,B 0,C 180,E1 -8350.061,E2 -8350.061} C_VEL
LIN {X 0,Y 457.588,Z 469.511,A -85,B 0,C 180,E1 -8350.952,E2 -8350.952} C_VEL
LIN {X 0,Y 456.609,Z 482.757,A -85,B 0,C 180,E1 -8352.072,E2 -8352.072} C_VEL
LIN {X 0,Y 455.821,Z 493.879,A -85,B 0,C 180,E1 -8353.197,E2 -8353.197} C_VEL
LIN {X 0,Y 454.912,Z 505.118,A -85,B 0,C 180,E1 -8354.544,E2 -8354.544} C_VEL
LIN {X 0,Y 454.114,Z 516.034,A -85,B 0,C 180,E1 -8356.121,E2 -8356.121} C_VEL
LIN {X 0,Y 453.489,Z 524.985,A -85,B 0,C 180,E1 -8357.668,E2 -8357.668} C_VEL
LIN {X 0,Y 453.148,Z 532.691,A -85,B 0,C 180,E1 -8359.274,E2 -8359.274} C_VEL
LIN {X 0,Y 452.777,Z 539.743,A -85,B 0,C 180,E1 -8361.071,E2 -8361.071} C_VEL
LIN {X 0,Y 452.646,Z 545.296,A -85,B 0,C 180,E1 -8362.865,E2 -8362.865} C_VEL
LIN {X 0,Y 452.52,Z 549.494,A -85,B 0,C 180,E1 -8364.654,E2 -8364.654} C_VEL
LIN {X 0,Y 452.498,Z 552.44,A -85,B 0,C 180,E1 -8366.439,E2 -8366.439} C_VEL
LIN {X 0,Y 452.472,Z 554.196,A -85,B 0,C 180,E1 -8368.22,E2 -8368.22} C_VEL
LIN {X 0,Y 452.461,Z 554.798,A -85,B 0,C 180,E1 -8370,E2 -8370} C_VEL
LIN {X 0,Y 452.473,Z 554.194,A -85,B 0,C 180,E1 -8371.781,E2 -8371.781} C_VEL
LIN {X 0,Y 452.498,Z 552.434,A -85,B 0,C 180,E1 -8373.562,E2 -8373.562} C_VEL
LIN {X 0,Y 452.544,Z 549.491,A -85,B 0,C 180,E1 -8375.347,E2 -8375.347} C_VEL
LIN {X 0,Y 452.648,Z 545.298,A -85,B 0,C 180,E1 -8377.136,E2 -8377.136} C_VEL
LIN {X 0,Y 452.777,Z 539.74,A -85,B 0,C 180,E1 -8378.93,E2 -8378.93} C_VEL
LIN {X 0,Y 453.15,Z 532.68,A -85,B 0,C 180,E1 -8380.726,E2 -8380.726} C_VEL
LIN {X 0,Y 453.526,Z 524.017,A -85,B 0,C 180,E1 -8382.507,E2 -8382.507} C_VEL
LIN {X 0,Y 454.228,Z 514.575,A -85,B 0,C 180,E1 -8384.105,E2 -8384.105} C_VEL
LIN {X 0,Y 454.887,Z 505.104,A -85,B 0,C 180,E1 -8385.457,E2 -8385.457} C_VEL
LIN {X 0,Y 455.865,Z 492.84,A -85,B 0,C 180,E1 -8386.918,E2 -8386.918} C_VEL
LIN {X 0,Y 456.785,Z 480.339,A -85,B 0,C 180,E1 -8388.154,E2 -8388.154} C_VEL
LIN {X 0,Y 457.834,Z 466.524,A -85,B 0,C 180,E1 -8389.271,E2 -8389.271} C_VEL
LIN {X 0,Y 458.814,Z 452.97,A -85,B 0,C 180,E1 -8390.161,E2 -8390.161} C_VEL
LIN {X 0,Y 459.59,Z 438.066,A -85,B 0,C 180,E1 -8390.938,E2 -8390.938} C_VEL
LIN {X 0,Y 459.993,Z 428.545,A -85,B 0,C 180,E1 -8391.329,E2 -8391.329} C_VEL
LIN {X 0,Y 456.813,Z 412.764,A -85,B 0,C 180,E1 -8392.001,E2 -8392.001} C_VEL
LIN {X 0,Y 453.223,Z 397.831,A -85,B 0,C 180,E1 -8392.518,E2 -8392.518} C_VEL
LIN {X 0,Y 453.538,Z 389.687,A -85,B 0,C 180,E1 -8396.004,E2 -8396.004} C_VEL
LIN {X 0,Y 453.852,Z 382.305,A -85,B 0,C 180,E1 -8399.195,E2 -8399.195} C_VEL
LIN {X 0,Y 454.172,Z 375.29,A -85,B 0,C 180,E1 -8402.267,E2 -8402.267} C_VEL
LIN {X 0,Y 454.536,Z 368.309,A -85,B 0,C 180,E1 -8405.438,E2 -8405.438} C_VEL
LIN {X 0,Y 454.803,Z 362.56,A -85,B 0,C 180,E1 -8408.179,E2 -8408.179} C_VEL
LIN {X 0,Y 455.175,Z 357.212,A -85,B 0,C 180,E1 -8410.837,E2 -8410.837} C_VEL
LIN {X 0,Y 454.928,Z 353.463,A -85,B 0,C 180,E1 -8412.824,E2 -8412.824} C_VEL
LIN {X 0,Y 454.104,Z 348.177,A -85,B 0,C 180,E1 -8415.857,E2 -8415.857} C_VEL
LIN {X 0,Y 453.479,Z 344.624,A -85,B 0,C 180,E1 -8418.065,E2 -8418.065} C_VEL
LIN {X 0,Y 453.512,Z 344.622,A -85,B 0,C 180,E1 -8420.791,E2 -8420.791} C_VEL
LIN {X 0,Y 453.46,Z 344.629,A -85,B 0,C 180,E1 -8423.918,E2 -8423.918} C_VEL
LIN {X 0,Y 453.485,Z 344.624,A -85,B 0,C 180,E1 -8427.151,E2 -8427.151} C_VEL
LIN {X 0,Y 453.477,Z 344.623,A -85,B 0,C 180,E1 -8430.269,E2 -8430.269} C_VEL
LIN {X 0,Y 453.509,Z 344.619,A -85,B 0,C 180,E1 -8433.294,E2 -8433.294} C_VEL
LIN {X 0,Y 453.505,Z 344.619,A -85,B 0,C 180,E1 -8436.239,E2 -8436.239} C_VEL
LIN {X 0,Y 453.485,Z 344.622,A -85,B 0,C 180,E1 -8439.118,E2 -8439.118} C_VEL
LIN {X 0,Y 453.515,Z 344.619,A -85,B 0,C 180,E1 -8441.945,E2 -8441.945} C_VEL
LIN {X 0,Y 453.543,Z 344.619,A -85,B 0,C 180,E1 -8444.727,E2 -8444.727} C_VEL
LIN {X 0,Y 453.563,Z 344.614,A -85,B 0,C 180,E1 -8448.379,E2 -8448.379} C_VEL
LIN {X 0,Y 453.655,Z 344.604,A -85,B 0,C 180,E1 -8451.985,E2 -8451.985} C_VEL
LIN {X 0,Y 453.674,Z 344.598,A -85,B 0,C 180,E1 -8454.667,E2 -8454.667} C_VEL
LIN {X 0,Y 453.768,Z 344.586,A -85,B 0,C 180,E1 -8457.337,E2 -8457.337} C_VEL
LIN {X 0,Y 453.826,Z 344.58,A -85,B 0,C 180,E1 -8460,E2 -8460} C_VEL
LIN {X 0,Y 453.768,Z 344.588,A -85,B 0,C 180,E1 -8462.663,E2 -8462.663} C_VEL
LIN {X 0,Y 453.682,Z 344.596,A -85,B 0,C 180,E1 -8466.225,E2 -8466.225} C_VEL
LIN {X 0,Y 453.596,Z 344.612,A -85,B 0,C 180,E1 -8468.913,E2 -8468.913} C_VEL
LIN {X 0,Y 453.567,Z 344.595,A -85,B 0,C 180,E1 -8472.529,E2 -8472.529} C_VEL
LIN {X 0,Y 453.548,Z 344.613,A -85,B 0,C 180,E1 -8476.196,E2 -8476.196} C_VEL
LIN {X 0,Y 453.524,Z 344.611,A -85,B 0,C 180,E1 -8479.041,E2 -8479.041} C_VEL
LIN {X 0,Y 453.48,Z 344.617,A -85,B 0,C 180,E1 -8481.836,E2 -8481.836} C_VEL
LIN {X 0,Y 453.504,Z 344.618,A -85,B 0,C 180,E1 -8484.735,E2 -8484.735} C_VEL
LIN {X 0,Y 453.536,Z 344.607,A -85,B 0,C 180,E1 -8487.96,E2 -8487.96} C_VEL
LIN {X 0,Y 453.469,Z 344.625,A -85,B 0,C 180,E1 -8491.525,E2 -8491.525} C_VEL
LIN {X 0,Y 453.492,Z 344.619,A -85,B 0,C 180,E1 -8494.777,E2 -8494.777} C_VEL
LIN {X 0,Y 453.476,Z 344.624,A -85,B 0,C 180,E1 -8498.311,E2 -8498.311} C_VEL
LIN {X 0,Y 453.497,Z 344.622,A -85,B 0,C 180,E1 -8500.609,E2 -8500.609} C_VEL
LIN {X 0,Y 453.459,Z 344.626,A -85,B 0,C 180,E1 -8503.244,E2 -8503.244} C_VEL
LIN {X 0,Y 453.468,Z 344.628,A -85,B 0,C 180,E1 -8505.779,E2 -8505.779} C_VEL
LIN {X 0,Y 453.415,Z 344.634,A -85,B 0,C 180,E1 -8508.202,E2 -8508.202} C_VEL
LIN {X 0,Y 453.169,Z 344.665,A -85,B 0,C 180,E1 -8510.844,E2 -8510.844} C_VEL
LIN {X 0,Y 453.1,Z 344.847,A -85,B 0,C 180,E1 -8511.652,E2 -8511.652} C_VEL
LIN {X 0,Y 453.069,Z 347.639,A -85,B 0,C 180,E1 -8514.974,E2 -8514.974} C_VEL
LIN {X 0,Y 452.954,Z 350.396,A -85,B 0,C 180,E1 -8518.16,E2 -8518.16} C_VEL
LIN {X 0,Y 452.903,Z 353.161,A -85,B 0,C 180,E1 -8521.246,E2 -8521.246} C_VEL
LIN {X 0,Y 452.822,Z 355.984,A -85,B 0,C 180,E1 -8524.242,E2 -8524.242} C_VEL
LIN {X 0,Y 452.727,Z 359.31,A -85,B 0,C 180,E1 -8527.552,E2 -8527.552} C_VEL
LIN {X 0,Y 455.11,Z 366.588,A -85,B 0,C 180,E1 -8527.834,E2 -8527.834} C_VEL
LIN {X 0,Y 459.849,Z 381.708,A -85,B 0,C 180,E1 -8528.523,E2 -8528.523} C_VEL
LIN {X 0,Y 460.605,Z 384.874,A -85,B 0,C 180,E1 -8528.683,E2 -8528.683} C_VEL
LIN {X 0,Y 459.96,Z 400.265,A -85,B 0,C 180,E1 -8529.345,E2 -8529.345} C_VEL
LIN {X 0,Y 459.202,Z 413.599,A -85,B 0,C 180,E1 -8530.09,E2 -8530.09} C_VEL
LIN {X 0,Y 458.403,Z 426.495,A -85,B 0,C 180,E1 -8530.986,E2 -8530.986} C_VEL
LIN {X 0,Y 457.474,Z 438.503,A -85,B 0,C 180,E1 -8531.99,E2 -8531.99} C_VEL
LIN {X 0,Y 456.497,Z 450.678,A -85,B 0,C 180,E1 -8533.222,E2 -8533.222} C_VEL
LIN {X 0,Y 455.613,Z 461.758,A -85,B 0,C 180,E1 -8534.568,E2 -8534.568} C_VEL
LIN {X 0,Y 455.448,Z 463.679,A -85,B 0,C 180,E1 -8534.833,E2 -8534.833} C_VEL
LIN {X 0,Y 454.521,Z 467.696,A -85,B 0,C 180,E1 -8535.375,E2 -8535.375} C_VEL
LIN {X 0,Y 451.202,Z 473.964,A -85,B 0,C 180,E1 -8536.247,E2 -8536.247} C_VEL
LIN {X 0,Y 447.924,Z 479.858,A -85,B 0,C 180,E1 -8537.174,E2 -8537.174} C_VEL
LIN {X 0,Y 447.074,Z 483.119,A -85,B 0,C 180,E1 -8537.794,E2 -8537.794} C_VEL
LIN {X 0,Y 446.438,Z 491.029,A -85,B 0,C 180,E1 -8539.569,E2 -8539.569} C_VEL
LIN {X 0,Y 446.039,Z 497.548,A -85,B 0,C 180,E1 -8541.391,E2 -8541.391} C_VEL
LIN {X 0,Y 445.813,Z 501.486,A -85,B 0,C 180,E1 -8542.754,E2 -8542.754} C_VEL
LIN {X 0,Y 445.588,Z 505.577,A -85,B 0,C 180,E1 -8544.569,E2 -8544.569} C_VEL
LIN {X 0,Y 445.56,Z 508.448,A -85,B 0,C 180,E1 -8546.382,E2 -8546.382} C_VEL
LIN {X 0,Y 445.453,Z 510.181,A -85,B 0,C 180,E1 -8548.191,E2 -8548.191} C_VEL
LIN {X 0,Y 445.398,Z 510.788,A -85,B 0,C 180,E1 -8550,E2 -8550} C_VEL
LIN {X 0,Y 445.454,Z 510.231,A -85,B 0,C 180,E1 -8551.808,E2 -8551.808} C_VEL
LIN {X 0,Y 445.56,Z 508.565,A -85,B 0,C 180,E1 -8553.617,E2 -8553.617} C_VEL
LIN {X 0,Y 445.584,Z 505.758,A -85,B 0,C 180,E1 -8555.43,E2 -8555.43} C_VEL
LIN {X 0,Y 445.809,Z 501.728,A -85,B 0,C 180,E1 -8557.245,E2 -8557.245} C_VEL
LIN {X 0,Y 446.099,Z 496.386,A -85,B 0,C 180,E1 -8559.064,E2 -8559.064} C_VEL
LIN {X 0,Y 446.503,Z 489.575,A -85,B 0,C 180,E1 -8560.887,E2 -8560.887} C_VEL
LIN {X 0,Y 447.114,Z 482.239,A -85,B 0,C 180,E1 -8562.481,E2 -8562.481} C_VEL
LIN {X 0,Y 447.783,Z 473.4,A -85,B 0,C 180,E1 -8564.079,E2 -8564.079} C_VEL
LIN {X 0,Y 448.571,Z 464.378,A -85,B 0,C 180,E1 -8565.447,E2 -8565.447} C_VEL
LIN {X 0,Y 449.447,Z 453.731,A -85,B 0,C 180,E1 -8566.815,E2 -8566.815} C_VEL
LIN {X 0,Y 450.426,Z 442.918,A -85,B 0,C 180,E1 -8567.982,E2 -8567.982} C_VEL
LIN {X 0,Y 451.376,Z 430.797,A -85,B 0,C 180,E1 -8569.085,E2 -8569.085} C_VEL
LIN {X 0,Y 452.312,Z 417.1,A -85,B 0,C 180,E1 -8570.107,E2 -8570.107} C_VEL
LIN {X 0,Y 453.202,Z 403.909,A -85,B 0,C 180,E1 -8570.895,E2 -8570.895} C_VEL
LIN {X 0,Y 453.819,Z 390.408,A -85,B 0,C 180,E1 -8571.534,E2 -8571.534} C_VEL
LIN {X 0,Y 453.819,Z 385.452,A -85,B 0,C 180,E1 -8571.735,E2 -8571.735} C_VEL
LIN {X 0,Y 449.373,Z 370.703,A -85,B 0,C 180,E1 -8572.457,E2 -8572.457} C_VEL
LIN {X 0,Y 445.653,Z 359.622,A -85,B 0,C 180,E1 -8572.921,E2 -8572.921} C_VEL
LIN {X 0,Y 445.757,Z 356.579,A -85,B 0,C 180,E1 -8576.014,E2 -8576.014} C_VEL
LIN {X 0,Y 445.842,Z 353.557,A -85,B 0,C 180,E1 -8579.252,E2 -8579.252} C_VEL
LIN {X 0,Y 445.918,Z 350.794,A -85,B 0,C 180,E1 -8582.402,E2 -8582.402} C_VEL
LIN {X 0,Y 446.007,Z 348.001,A -85,B 0,C 180,E1 -8585.663,E2 -8585.663} C_VEL
LIN {X 0,Y 446.055,Z 346.021,A -85,B 0,C 180,E1 -8588.02,E2 -8588.02} C_VEL
LIN {X 0,Y 446.164,Z 345.537,A -85,B 0,C 180,E1 -8589.479,E2 -8589.479} C_VEL
LIN {X 0,Y 446.371,Z 345.505,A -85,B 0,C 180,E1 -8592.268,E2 -8592.268} C_VEL
LIN {X 0,Y 446.452,Z 345.498,A -85,B 0,C 180,E1 -8595.103,E2 -8595.103} C_VEL
LIN {X 0,Y 446.427,Z 345.501,A -85,B 0,C 180,E1 -8598.609,E2 -8598.609} C_VEL
LIN {X 0,Y 446.46,Z 345.498,A -85,B 0,C 180,E1 -8600.974,E2 -8600.974} C_VEL
LIN {X 0,Y 446.42,Z 345.502,A -85,B 0,C 180,E1 -8604.374,E2 -8604.374} C_VEL
LIN {X 0,Y 446.421,Z 345.495,A -85,B 0,C 180,E1 -8607.638,E2 -8607.638} C_VEL
LIN {X 0,Y 446.468,Z 345.495,A -85,B 0,C 180,E1 -8610.792,E2 -8610.792} C_VEL
LIN {X 0,Y 446.476,Z 345.487,A -85,B 0,C 180,E1 -8613.848,E2 -8613.848} C_VEL
LIN {X 0,Y 446.428,Z 345.5,A -85,B 0,C 180,E1 -8616.823,E2 -8616.823} C_VEL
LIN {X 0,Y 446.443,Z 345.485,A -85,B 0,C 180,E1 -8619.737,E2 -8619.737} C_VEL
LIN {X 0,Y 446.462,Z 345.496,A -85,B 0,C 180,E1 -8622.597,E2 -8622.597} C_VEL
LIN {X 0,Y 446.468,Z 345.488,A -85,B 0,C 180,E1 -8625.412,E2 -8625.412} C_VEL
LIN {X 0,Y 446.538,Z 345.481,A -85,B 0,C 180,E1 -8628.193,E2 -8628.193} C_VEL
LIN {X 0,Y 446.598,Z 345.478,A -85,B 0,C 180,E1 -8631.858,E2 -8631.858} C_VEL
LIN {X 0,Y 446.644,Z 345.474,A -85,B 0,C 180,E1 -8634.582,E2 -8634.582} C_VEL
LIN {X 0,Y 446.707,Z 345.469,A -85,B 0,C 180,E1 -8637.295,E2 -8637.295} C_VEL
LIN {X 0,Y 446.792,Z 345.458,A -85,B 0,C 180,E1 -8640,E2 -8640} C_VEL
LIN {X 0,Y 446.708,Z 345.466,A -85,B 0,C 180,E1 -8642.705,E2 -8642.705} C_VEL
LIN {X 0,Y 446.645,Z 345.477,A -85,B 0,C 180,E1 -8646.324,E2 -8646.324} C_VEL
LIN {X 0,Y 446.536,Z 345.489,A -85,B 0,C 180,E1 -8649.055,E2 -8649.055} C_VEL
LIN {X 0,Y 446.519,Z 345.489,A -85,B 0,C 180,E1 -8652.73,E2 -8652.73} C_VEL
LIN {X 0,Y 446.494,Z 345.491,A -85,B 0,C 180,E1 -8656.228,E2 -8656.228} C_VEL
LIN {X 0,Y 446.467,Z 345.496,A -85,B 0,C 180,E1 -8659.303,E2 -8659.303} C_VEL
LIN {X 0,Y 446.416,Z 345.502,A -85,B 0,C 180,E1 -8662.2,E2 -8662.2} C_VEL
LIN {X 0,Y 446.455,Z 345.499,A -85,B 0,C 180,E1 -8665.152,E2 -8665.152} C_VEL
LIN {X 0,Y 446.482,Z 345.496,A -85,B 0,C 180,E1 -8668.179,E2 -8668.179} C_VEL
LIN {X 0,Y 446.418,Z 345.503,A -85,B 0,C 180,E1 -8671.3,E2 -8671.3} C_VEL
LIN {X 0,Y 446.428,Z 345.502,A -85,B 0,C 180,E1 -8674.523,E2 -8674.523} C_VEL
LIN {X 0,Y 446.428,Z 345.503,A -85,B 0,C 180,E1 -8678.082,E2 -8678.082} C_VEL
LIN {X 0,Y 446.424,Z 345.504,A -85,B 0,C 180,E1 -8680.918,E2 -8680.918} C_VEL
LIN {X 0,Y 446.452,Z 345.616,A -85,B 0,C 180,E1 -8681.622,E2 -8681.622} C_VEL
LIN {X 0,Y 447.397,Z 350.994,A -85,B 0,C 180,E1 -8684.982,E2 -8684.982} C_VEL
LIN {X 0,Y 448.084,Z 355.605,A -85,B 0,C 180,E1 -8687.59,E2 -8687.59} C_VEL
LIN {X 0,Y 448.183,Z 358.999,A -85,B 0,C 180,E1 -8689.408,E2 -8689.408} C_VEL
LIN {X 0,Y 447.777,Z 364.699,A -85,B 0,C 180,E1 -8692.258,E2 -8692.258} C_VEL
LIN {X 0,Y 447.511,Z 369.895,A -85,B 0,C 180,E1 -8694.75,E2 -8694.75} C_VEL
LIN {X 0,Y 447.117,Z 377.09,A -85,B 0,C 180,E1 -8698.081,E2 -8698.081} C_VEL
LIN {X 0,Y 446.726,Z 384.35,A -85,B 0,C 180,E1 -8701.327,E2 -8701.327} C_VEL
LIN {X 0,Y 446.361,Z 392.344,A -85,B 0,C 180,E1 -8704.842,E2 -8704.842} C_VEL
LIN {X 0,Y 446.158,Z 397.523,A -85,B 0,C 180,E1 -8707.119,E2 -8707.119} C_VEL
LIN {X 0,Y 450.385,Z 414.943,A -85,B 0,C 180,E1 -8707.733,E2 -8707.733} C_VEL
LIN {X 0,Y 453.36,Z 429.863,A -85,B 0,C 180,E1 -8708.408,E2 -8708.408} C_VEL
LIN {X 0,Y 452.626,Z 444.532,A -85,B 0,C 180,E1 -8709.077,E2 -8709.077} C_VEL
LIN {X 0,Y 451.705,Z 458.037,A -85,B 0,C 180,E1 -8709.865,E2 -8709.865} C_VEL
LIN {X 0,Y 450.713,Z 470.597,A -85,B 0,C 180,E1 -8710.768,E2 -8710.768} C_VEL
LIN {X 0,Y 449.687,Z 483.708,A -85,B 0,C 180,E1 -8711.916,E2 -8711.916} C_VEL
LIN {X 0,Y 448.778,Z 495.786,A -85,B 0,C 180,E1 -8713.194,E2 -8713.194} C_VEL
LIN {X 0,Y 447.821,Z 506.412,A -85,B 0,C 180,E1 -8714.527,E2 -8714.527} C_VEL
LIN {X 0,Y 447.015,Z 517.052,A -85,B 0,C 180,E1 -8716.128,E2 -8716.128} C_VEL
LIN {X 0,Y 446.423,Z 526.248,A -85,B 0,C 180,E1 -8717.797,E2 -8717.797} C_VEL
LIN {X 0,Y 445.959,Z 534.232,A -85,B 0,C 180,E1 -8719.559,E2 -8719.559} C_VEL
LIN {X 0,Y 445.65,Z 540.9,A -85,B 0,C 180,E1 -8721.384,E2 -8721.384} C_VEL
LIN {X 0,Y 445.498,Z 546.123,A -85,B 0,C 180,E1 -8723.205,E2 -8723.205} C_VEL
LIN {X 0,Y 445.438,Z 549.146,A -85,B 0,C 180,E1 -8724.568,E2 -8724.568} C_VEL
LIN {X 0,Y 445.396,Z 552.091,A -85,B 0,C 180,E1 -8726.382,E2 -8726.382} C_VEL
LIN {X 0,Y 445.388,Z 553.849,A -85,B 0,C 180,E1 -8728.192,E2 -8728.192} C_VEL
LIN {X 0,Y 445.397,Z 554.452,A -85,B 0,C 180,E1 -8730,E2 -8730} C_VEL
LIN {X 0,Y 445.388,Z 553.846,A -85,B 0,C 180,E1 -8731.809,E2 -8731.809} C_VEL
LIN {X 0,Y 445.397,Z 552.085,A -85,B 0,C 180,E1 -8733.619,E2 -8733.619} C_VEL
LIN {X 0,Y 445.463,Z 549.142,A -85,B 0,C 180,E1 -8735.432,E2 -8735.432} C_VEL
LIN {X 0,Y 445.572,Z 544.948,A -85,B 0,C 180,E1 -8737.25,E2 -8737.25} C_VEL
LIN {X 0,Y 445.697,Z 539.388,A -85,B 0,C 180,E1 -8739.073,E2 -8739.073} C_VEL
LIN {X 0,Y 446.12,Z 532.328,A -85,B 0,C 180,E1 -8740.897,E2 -8740.897} C_VEL
LIN {X 0,Y 446.482,Z 524.264,A -85,B 0,C 180,E1 -8742.597,E2 -8742.597} C_VEL
LIN {X 0,Y 447.139,Z 515.673,A -85,B 0,C 180,E1 -8744.101,E2 -8744.101} C_VEL
LIN {X 0,Y 447.965,Z 504.75,A -85,B 0,C 180,E1 -8745.702,E2 -8745.702} C_VEL
LIN {X 0,Y 449.002,Z 492.623,A -85,B 0,C 180,E1 -8747.17,E2 -8747.17} C_VEL
LIN {X 0,Y 449.975,Z 479.985,A -85,B 0,C 180,E1 -8748.438,E2 -8748.438} C_VEL
LIN {X 0,Y 451.094,Z 466.17,A -85,B 0,C 180,E1 -8749.571,E2 -8749.571} C_VEL
LIN {X 0,Y 452.127,Z 452.616,A -85,B 0,C 180,E1 -8750.472,E2 -8750.472} C_VEL
LIN {X 0,Y 452.93,Z 437.796,A -85,B 0,C 180,E1 -8751.256,E2 -8751.256} C_VEL
LIN {X 0,Y 453.246,Z 429.427,A -85,B 0,C 180,E1 -8751.613,E2 -8751.613} C_VEL
LIN {X 0,Y 450.103,Z 413.739,A -85,B 0,C 180,E1 -8752.311,E2 -8752.311} C_VEL
LIN {X 0,Y 446.159,Z 397.513,A -85,B 0,C 180,E1 -8752.882,E2 -8752.882} C_VEL
LIN {X 0,Y 446.477,Z 389.931,A -85,B 0,C 180,E1 -8756.203,E2 -8756.203} C_VEL
LIN {X 0,Y 446.841,Z 382.117,A -85,B 0,C 180,E1 -8759.655,E2 -8759.655} C_VEL
LIN {X 0,Y 447.269,Z 373.868,A -85,B 0,C 180,E1 -8763.365,E2 -8763.365} C_VEL
LIN {X 0,Y 447.674,Z 366.916,A -85,B 0,C 180,E1 -8766.624,E2 -8766.624} C_VEL
LIN {X 0,Y 448.045,Z 360.077,A -85,B 0,C 180,E1 -8770.025,E2 -8770.025} C_VEL
LIN {X 0,Y 448.156,Z 356.686,A -85,B 0,C 180,E1 -8771.797,E2 -8771.797} C_VEL
LIN {X 0,Y 447.578,Z 352.041,A -85,B 0,C 180,E1 -8774.402,E2 -8774.402} C_VEL
LIN {X 0,Y 446.644,Z 346.647,A -85,B 0,C 180,E1 -8777.694,E2 -8777.694} C_VEL
LIN {X 0,Y 446.425,Z 345.503,A -85,B 0,C 180,E1 -8778.492,E2 -8778.492} C_VEL
LIN {X 0,Y 446.459,Z 345.501,A -85,B 0,C 180,E1 -8780.975,E2 -8780.975} C_VEL
LIN {X 0,Y 446.424,Z 345.505,A -85,B 0,C 180,E1 -8784.374,E2 -8784.374} C_VEL
LIN {X 0,Y 446.424,Z 345.503,A -85,B 0,C 180,E1 -8787.639,E2 -8787.639} C_VEL
LIN {X 0,Y 446.452,Z 345.501,A -85,B 0,C 180,E1 -8790.791,E2 -8790.791} C_VEL
LIN {X 0,Y 446.48,Z 345.498,A -85,B 0,C 180,E1 -8793.849,E2 -8793.849} C_VEL
LIN {X 0,Y 446.431,Z 345.504,A -85,B 0,C 180,E1 -8796.824,E2 -8796.824} C_VEL
LIN {X 0,Y 446.447,Z 345.5,A -85,B 0,C 180,E1 -8799.737,E2 -8799.737} C_VEL
LIN {X 0,Y 446.467,Z 345.497,A -85,B 0,C 180,E1 -8802.597,E2 -8802.597} C_VEL
LIN {X 0,Y 446.473,Z 345.497,A -85,B 0,C 180,E1 -8805.413,E2 -8805.413} C_VEL
LIN {X 0,Y 446.521,Z 345.491,A -85,B 0,C 180,E1 -8808.193,E2 -8808.193} C_VEL
LIN {X 0,Y 446.604,Z 345.481,A -85,B 0,C 180,E1 -8811.858,E2 -8811.858} C_VEL
LIN {X 0,Y 446.648,Z 345.473,A -85,B 0,C 180,E1 -8814.583,E2 -8814.583} C_VEL
LIN {X 0,Y 446.712,Z 345.465,A -85,B 0,C 180,E1 -8817.295,E2 -8817.295} C_VEL
LIN {X 0,Y 446.796,Z 345.456,A -85,B 0,C 180,E1 -8820,E2 -8820} C_VEL
LIN {X 0,Y 446.712,Z 345.467,A -85,B 0,C 180,E1 -8822.705,E2 -8822.705} C_VEL
LIN {X 0,Y 446.651,Z 345.471,A -85,B 0,C 180,E1 -8826.324,E2 -8826.324} C_VEL
LIN {X 0,Y 446.542,Z 345.489,A -85,B 0,C 180,E1 -8829.055,E2 -8829.055} C_VEL
LIN {X 0,Y 446.525,Z 345.471,A -85,B 0,C 180,E1 -8832.73,E2 -8832.73} C_VEL
LIN {X 0,Y 446.5,Z 345.491,A -85,B 0,C 180,E1 -8836.228,E2 -8836.228} C_VEL
LIN {X 0,Y 446.473,Z 345.489,A -85,B 0,C 180,E1 -8839.303,E2 -8839.303} C_VEL
LIN {X 0,Y 446.421,Z 345.496,A -85,B 0,C 180,E1 -8842.2,E2 -8842.2} C_VEL
LIN {X 0,Y 446.447,Z 345.497,A -85,B 0,C 180,E1 -8845.153,E2 -8845.153} C_VEL
LIN {X 0,Y 446.488,Z 345.485,A -85,B 0,C 180,E1 -8848.179,E2 -8848.179} C_VEL
LIN {X 0,Y 446.422,Z 345.501,A -85,B 0,C 180,E1 -8851.775,E2 -8851.775} C_VEL
LIN {X 0,Y 446.433,Z 345.495,A -85,B 0,C 180,E1 -8854.523,E2 -8854.523} C_VEL
LIN {X 0,Y 446.434,Z 345.503,A -85,B 0,C 180,E1 -8858.082,E2 -8858.082} C_VEL
LIN {X 0,Y 446.43,Z 345.504,A -85,B 0,C 180,E1 -8860.918,E2 -8860.918} C_VEL
LIN {X 0,Y 446.405,Z 345.508,A -85,B 0,C 180,E1 -8863.846,E2 -8863.846} C_VEL
LIN {X 0,Y 446.429,Z 345.503,A -85,B 0,C 180,E1 -8866.4,E2 -8866.4} C_VEL
LIN {X 0,Y 446.285,Z 345.523,A -85,B 0,C 180,E1 -8869.104,E2 -8869.104} C_VEL
LIN {X 0,Y 446.108,Z 345.544,A -85,B 0,C 180,E1 -8870.938,E2 -8870.938} C_VEL
LIN {X 0,Y 446.055,Z 346.028,A -85,B 0,C 180,E1 -8872.085,E2 -8872.085} C_VEL
LIN {X 0,Y 446.003,Z 348.828,A -85,B 0,C 180,E1 -8875.439,E2 -8875.439} C_VEL
LIN {X 0,Y 445.916,Z 351.592,A -85,B 0,C 180,E1 -8878.66,E2 -8878.66} C_VEL
LIN {X 0,Y 445.834,Z 354.595,A -85,B 0,C 180,E1 -8881.978,E2 -8881.978} C_VEL
LIN {X 0,Y 445.737,Z 357.255,A -85,B 0,C 180,E1 -8884.804,E2 -8884.804} C_VEL
LIN {X 0,Y 445.661,Z 359.662,A -85,B 0,C 180,E1 -8887.18,E2 -8887.18} C_VEL
LIN {X 0,Y 451.038,Z 375.881,A -85,B 0,C 180,E1 -8887.872,E2 -8887.872} C_VEL
LIN {X 0,Y 454.003,Z 386.506,A -85,B 0,C 180,E1 -8888.408,E2 -8888.408} C_VEL
LIN {X 0,Y 453.32,Z 400.773,A -85,B 0,C 180,E1 -8889.036,E2 -8889.036} C_VEL
LIN {X 0,Y 452.535,Z 413.954,A -85,B 0,C 180,E1 -8889.784,E2 -8889.784} C_VEL
LIN {X 0,Y 451.696,Z 426.849,A -85,B 0,C 180,E1 -8890.693,E2 -8890.693} C_VEL
LIN {X 0,Y 450.722,Z 438.856,A -85,B 0,C 180,E1 -8891.711,E2 -8891.711} C_VEL
LIN {X 0,Y 449.691,Z 451.031,A -85,B 0,C 180,E1 -8892.96,E2 -8892.96} C_VEL
LIN {X 0,Y 448.764,Z 462.11,A -85,B 0,C 180,E1 -8894.327,E2 -8894.327} C_VEL
LIN {X 0,Y 447.835,Z 472.866,A -85,B 0,C 180,E1 -8895.921,E2 -8895.921} C_VEL
LIN {X 0,Y 447.146,Z 481.781,A -85,B 0,C 180,E1 -8897.519,E2 -8897.519} C_VEL
LIN {X 0,Y 447.074,Z 483.119,A -85,B 0,C 180,E1 -8897.794,E2 -8897.794} C_VEL
LIN {X 0,Y 446.24,Z 486.281,A -85,B 0,C 180,E1 -8898.432,E2 -8898.432} C_VEL
LIN {X 0,Y 443.028,Z 491.119,A -85,B 0,C 180,E1 -8899.467,E2 -8899.467} C_VEL
LIN {X 0,Y 439.816,Z 495.507,A -85,B 0,C 180,E1 -8900.546,E2 -8900.546} C_VEL
LIN {X 0,Y 438.994,Z 497.868,A -85,B 0,C 180,E1 -8901.242,E2 -8901.242} C_VEL
LIN {X 0,Y 438.757,Z 501.836,A -85,B 0,C 180,E1 -8902.637,E2 -8902.637} C_VEL
LIN {X 0,Y 438.533,Z 505.926,A -85,B 0,C 180,E1 -8904.482,E2 -8904.482} C_VEL
LIN {X 0,Y 438.478,Z 508.796,A -85,B 0,C 180,E1 -8906.324,E2 -8906.324} C_VEL
LIN {X 0,Y 438.37,Z 510.529,A -85,B 0,C 180,E1 -8908.162,E2 -8908.162} C_VEL
LIN {X 0,Y 438.32,Z 511.135,A -85,B 0,C 180,E1 -8910,E2 -8910} C_VEL
LIN {X 0,Y 438.37,Z 510.578,A -85,B 0,C 180,E1 -8911.837,E2 -8911.837} C_VEL
LIN {X 0,Y 438.477,Z 508.912,A -85,B 0,C 180,E1 -8913.676,E2 -8913.676} C_VEL
LIN {X 0,Y 438.529,Z 506.104,A -85,B 0,C 180,E1 -8915.518,E2 -8915.518} C_VEL
LIN {X 0,Y 438.754,Z 502.076,A -85,B 0,C 180,E1 -8917.362,E2 -8917.362} C_VEL
LIN {X 0,Y 439.075,Z 496.733,A -85,B 0,C 180,E1 -8919.21,E2 -8919.21} C_VEL
LIN {X 0,Y 439.509,Z 489.922,A -85,B 0,C 180,E1 -8921.062,E2 -8921.062} C_VEL
LIN {X 0,Y 440.163,Z 482.585,A -85,B 0,C 180,E1 -8922.682,E2 -8922.682} C_VEL
LIN {X 0,Y 440.867,Z 473.747,A -85,B 0,C 180,E1 -8924.305,E2 -8924.305} C_VEL
LIN {X 0,Y 441.718,Z 464.724,A -85,B 0,C 180,E1 -8925.692,E2 -8925.692} C_VEL
LIN {X 0,Y 442.624,Z 454.077,A -85,B 0,C 180,E1 -8927.082,E2 -8927.082} C_VEL
LIN {X 0,Y 443.736,Z 442.391,A -85,B 0,C 180,E1 -8928.352,E2 -8928.352} C_VEL
LIN {X 0,Y 444.797,Z 429.723,A -85,B 0,C 180,E1 -8929.498,E2 -8929.498} C_VEL
LIN {X 0,Y 445.819,Z 415.682,A -85,B 0,C 180,E1 -8930.533,E2 -8930.533} C_VEL
LIN {X 0,Y 446.779,Z 401.14,A -85,B 0,C 180,E1 -8931.377,E2 -8931.377} C_VEL
LIN {X 0,Y 447.253,Z 387.277,A -85,B 0,C 180,E1 -8932.011,E2 -8932.011} C_VEL
LIN {X 0,Y 443.047,Z 373.01,A -85,B 0,C 180,E1 -8932.741,E2 -8932.741} C_VEL
LIN {X 0,Y 438.75,Z 360.82,A -85,B 0,C 180,E1 -8933.274,E2 -8933.274} C_VEL
LIN {X 0,Y 438.629,Z 359.946,A -85,B 0,C 180,E1 -8933.332,E2 -8933.332} C_VEL
LIN {X 0,Y 438.711,Z 356.73,A -85,B 0,C 180,E1 -8936.65,E2 -8936.65} C_VEL
LIN {X 0,Y 438.771,Z 354.819,A -85,B 0,C 180,E1 -8938.719,E2 -8938.719} C_VEL
LIN {X 0,Y 438.853,Z 351.968,A -85,B 0,C 180,E1 -8941.922,E2 -8941.922} C_VEL
LIN {X 0,Y 438.962,Z 349.168,A -85,B 0,C 180,E1 -8945.196,E2 -8945.196} C_VEL
LIN {X 0,Y 438.999,Z 346.599,A -85,B 0,C 180,E1 -8948.33,E2 -8948.33} C_VEL
LIN {X 0,Y 439.284,Z 346.39,A -85,B 0,C 180,E1 -8951.241,E2 -8951.241} C_VEL
LIN {X 0,Y 439.403,Z 346.378,A -85,B 0,C 180,E1 -8954.728,E2 -8954.728} C_VEL
LIN {X 0,Y 439.394,Z 346.379,A -85,B 0,C 180,E1 -8957.795,E2 -8957.795} C_VEL
LIN {X 0,Y 439.435,Z 346.373,A -85,B 0,C 180,E1 -8960.228,E2 -8960.228} C_VEL
LIN {X 0,Y 439.376,Z 346.382,A -85,B 0,C 180,E1 -8963.713,E2 -8963.713} C_VEL
LIN {X 0,Y 439.371,Z 346.373,A -85,B 0,C 180,E1 -8967.054,E2 -8967.054} C_VEL
LIN {X 0,Y 439.395,Z 346.376,A -85,B 0,C 180,E1 -8970.275,E2 -8970.275} C_VEL
LIN {X 0,Y 439.432,Z 346.364,A -85,B 0,C 180,E1 -8973.588,E2 -8973.588} C_VEL
LIN {X 0,Y 439.385,Z 346.377,A -85,B 0,C 180,E1 -8976.429,E2 -8976.429} C_VEL
LIN {X 0,Y 439.387,Z 346.364,A -85,B 0,C 180,E1 -8979.397,E2 -8979.397} C_VEL
LIN {X 0,Y 439.43,Z 346.373,A -85,B 0,C 180,E1 -8982.309,E2 -8982.309} C_VEL
LIN {X 0,Y 439.446,Z 346.365,A -85,B 0,C 180,E1 -8985.174,E2 -8985.174} C_VEL
LIN {X 0,Y 439.506,Z 346.354,A -85,B 0,C 180,E1 -8988.002,E2 -8988.002} C_VEL
LIN {X 0,Y 439.546,Z 346.357,A -85,B 0,C 180,E1 -8991.726,E2 -8991.726} C_VEL
LIN {X 0,Y 439.62,Z 346.35,A -85,B 0,C 180,E1 -8994.496,E2 -8994.496} C_VEL
LIN {X 0,Y 439.635,Z 346.347,A -85,B 0,C 180,E1 -8998.168,E2 -8998.168} C_VEL
LIN {X 0,Y 439.762,Z 346.334,A -85,B 0,C 180,E1 -9000,E2 -9000} C_VEL
LIN {X 0,Y 439.655,Z 346.344,A -85,B 0,C 180,E1 -9002.749,E2 -9002.749} C_VEL
LIN {X 0,Y 439.616,Z 346.352,A -85,B 0,C 180,E1 -9006.425,E2 -9006.425} C_VEL
LIN {X 0,Y 439.498,Z 346.367,A -85,B 0,C 180,E1 -9009.202,E2 -9009.202} C_VEL
LIN {X 0,Y 439.463,Z 346.367,A -85,B 0,C 180,E1 -9012.938,E2 -9012.938} C_VEL
LIN {X 0,Y 439.445,Z 346.369,A -85,B 0,C 180,E1 -9016.349,E2 -9016.349} C_VEL
LIN {X 0,Y 439.4,Z 346.377,A -85,B 0,C 180,E1 -9019.626,E2 -9019.626} C_VEL
LIN {X 0,Y 439.363,Z 346.381,A -85,B 0,C 180,E1 -9022.575,E2 -9022.575} C_VEL
LIN {X 0,Y 439.403,Z 346.377,A -85,B 0,C 180,E1 -9025.585,E2 -9025.585} C_VEL
LIN {X 0,Y 439.423,Z 346.375,A -85,B 0,C 180,E1 -9028.673,E2 -9028.673} C_VEL
LIN {X 0,Y 439.38,Z 346.38,A -85,B 0,C 180,E1 -9032.033,E2 -9032.033} C_VEL
LIN {X 0,Y 439.394,Z 346.379,A -85,B 0,C 180,E1 -9035.341,E2 -9035.341} C_VEL
LIN {X 0,Y 439.388,Z 346.38,A -85,B 0,C 180,E1 -9038.594,E2 -9038.594} C_VEL
LIN {X 0,Y 439.41,Z 346.536,A -85,B 0,C 180,E1 -9041.261,E2 -9041.261} C_VEL
LIN {X 0,Y 440.333,Z 351.798,A -85,B 0,C 180,E1 -9044.609,E2 -9044.609} C_VEL
LIN {X 0,Y 441.012,Z 356.118,A -85,B 0,C 180,E1 -9047.143,E2 -9047.143} C_VEL
LIN {X 0,Y 441.205,Z 359.922,A -85,B 0,C 180,E1 -9049.225,E2 -9049.225} C_VEL
LIN {X 0,Y 440.706,Z 367.138,A -85,B 0,C 180,E1 -9052.878,E2 -9052.878} C_VEL
LIN {X 0,Y 440.32,Z 373.8,A -85,B 0,C 180,E1 -9056.096,E2 -9056.096} C_VEL
LIN {X 0,Y 439.933,Z 380.609,A -85,B 0,C 180,E1 -9059.256,E2 -9059.256} C_VEL
LIN {X 0,Y 439.525,Z 387.48,A -85,B 0,C 180,E1 -9062.374,E2 -9062.374} C_VEL
LIN {X 0,Y 439.218,Z 394.24,A -85,B 0,C 180,E1 -9065.416,E2 -9065.416} C_VEL
LIN {X 0,Y 439.11,Z 397.153,A -85,B 0,C 180,E1 -9066.721,E2 -9066.721} C_VEL
LIN {X 0,Y 443.577,Z 415.25,A -85,B 0,C 180,E1 -9067.392,E2 -9067.392} C_VEL
LIN {X 0,Y 446.502,Z 430.435,A -85,B 0,C 180,E1 -9068.096,E2 -9068.096} C_VEL
LIN {X 0,Y 445.908,Z 445.312,A -85,B 0,C 180,E1 -9068.807,E2 -9068.807} C_VEL
LIN {X 0,Y 444.849,Z 459.463,A -85,B 0,C 180,E1 -9069.662,E2 -9069.662} C_VEL
LIN {X 0,Y 443.757,Z 473.118,A -85,B 0,C 180,E1 -9070.695,E2 -9070.695} C_VEL
LIN {X 0,Y 442.688,Z 485.606,A -85,B 0,C 180,E1 -9071.847,E2 -9071.847} C_VEL
LIN {X 0,Y 441.736,Z 497.475,A -85,B 0,C 180,E1 -9073.164,E2 -9073.164} C_VEL
LIN {X 0,Y 440.745,Z 507.704,A -85,B 0,C 180,E1 -9074.509,E2 -9074.509} C_VEL
LIN {X 0,Y 439.923,Z 518.07,A -85,B 0,C 180,E1 -9076.136,E2 -9076.136} C_VEL
LIN {X 0,Y 439.368,Z 526.609,A -85,B 0,C 180,E1 -9077.746,E2 -9077.746} C_VEL
LIN {X 0,Y 438.929,Z 533.882,A -85,B 0,C 180,E1 -9079.39,E2 -9079.39} C_VEL
LIN {X 0,Y 438.562,Z 540.55,A -85,B 0,C 180,E1 -9081.244,E2 -9081.244} C_VEL
LIN {X 0,Y 438.413,Z 545.774,A -85,B 0,C 180,E1 -9083.095,E2 -9083.095} C_VEL
LIN {X 0,Y 438.342,Z 548.797,A -85,B 0,C 180,E1 -9084.48,E2 -9084.48} C_VEL
LIN {X 0,Y 438.296,Z 551.743,A -85,B 0,C 180,E1 -9086.323,E2 -9086.323} C_VEL
LIN {X 0,Y 438.308,Z 553.502,A -85,B 0,C 180,E1 -9088.163,E2 -9088.163} C_VEL
LIN {X 0,Y 438.305,Z 554.104,A -85,B 0,C 180,E1 -9090,E2 -9090} C_VEL
LIN {X 0,Y 438.308,Z 553.499,A -85,B 0,C 180,E1 -9091.838,E2 -9091.838} C_VEL
LIN {X 0,Y 438.298,Z 551.736,A -85,B 0,C 180,E1 -9093.678,E2 -9093.678} C_VEL
LIN {X 0,Y 438.367,Z 548.792,A -85,B 0,C 180,E1 -9095.52,E2 -9095.52} C_VEL
LIN {X 0,Y 438.487,Z 544.597,A -85,B 0,C 180,E1 -9097.367,E2 -9097.367} C_VEL
LIN {X 0,Y 438.627,Z 539.036,A -85,B 0,C 180,E1 -9099.22,E2 -9099.22} C_VEL
LIN {X 0,Y 439.095,Z 531.976,A -85,B 0,C 180,E1 -9101.074,E2 -9101.074} C_VEL
LIN {X 0,Y 439.543,Z 523.187,A -85,B 0,C 180,E1 -9102.936,E2 -9102.936} C_VEL
LIN {X 0,Y 440.284,Z 513.866,A -85,B 0,C 180,E1 -9104.561,E2 -9104.561} C_VEL
LIN {X 0,Y 441.037,Z 504.395,A -85,B 0,C 180,E1 -9105.955,E2 -9105.955} C_VEL
LIN {X 0,Y 442.058,Z 493.175,A -85,B 0,C 180,E1 -9107.342,E2 -9107.342} C_VEL
LIN {X 0,Y 443.062,Z 480.856,A -85,B 0,C 180,E1 -9108.617,E2 -9108.617} C_VEL
LIN {X 0,Y 444.231,Z 467.344,A -85,B 0,C 180,E1 -9109.766,E2 -9109.766} C_VEL
LIN {X 0,Y 445.287,Z 454.085,A -85,B 0,C 180,E1 -9110.68,E2 -9110.68} C_VEL
LIN {X 0,Y 446.192,Z 439.402,A -85,B 0,C 180,E1 -9111.493,E2 -9111.493} C_VEL
LIN {X 0,Y 446.675,Z 431.575,A -85,B 0,C 180,E1 -9111.842,E2 -9111.842} C_VEL
LIN {X 0,Y 443.762,Z 416.27,A -85,B 0,C 180,E1 -9112.562,E2 -9112.562} C_VEL
LIN {X 0,Y 440.024,Z 401.091,A -85,B 0,C 180,E1 -9113.139,E2 -9113.139} C_VEL
LIN {X 0,Y 439.109,Z 397.141,A -85,B 0,C 180,E1 -9113.28,E2 -9113.28} C_VEL
LIN {X 0,Y 439.439,Z 389.728,A -85,B 0,C 180,E1 -9116.603,E2 -9116.603} C_VEL
LIN {X 0,Y 439.788,Z 382.865,A -85,B 0,C 180,E1 -9119.696,E2 -9119.696} C_VEL
LIN {X 0,Y 440.251,Z 374.834,A -85,B 0,C 180,E1 -9123.386,E2 -9123.386} C_VEL
LIN {X 0,Y 440.587,Z 369,A -85,B 0,C 180,E1 -9126.172,E2 -9126.172} C_VEL
LIN {X 0,Y 440.984,Z 362.139,A -85,B 0,C 180,E1 -9129.605,E2 -9129.605} C_VEL
LIN {X 0,Y 441.192,Z 358.495,A -85,B 0,C 180,E1 -9131.523,E2 -9131.523} C_VEL
LIN {X 0,Y 440.68,Z 353.871,A -85,B 0,C 180,E1 -9134.138,E2 -9134.138} C_VEL
LIN {X 0,Y 439.79,Z 348.688,A -85,B 0,C 180,E1 -9137.316,E2 -9137.316} C_VEL
LIN {X 0,Y 439.406,Z 346.378,A -85,B 0,C 180,E1 -9138.922,E2 -9138.922} C_VEL
LIN {X 0,Y 439.387,Z 346.382,A -85,B 0,C 180,E1 -9141.606,E2 -9141.606} C_VEL
LIN {X 0,Y 439.404,Z 346.382,A -85,B 0,C 180,E1 -9144.845,E2 -9144.845} C_VEL
LIN {X 0,Y 439.375,Z 346.382,A -85,B 0,C 180,E1 -9148.14,E2 -9148.14} C_VEL
LIN {X 0,Y 439.435,Z 346.372,A -85,B 0,C 180,E1 -9151.598,E2 -9151.598} C_VEL
LIN {X 0,Y 439.403,Z 346.377,A -85,B 0,C 180,E1 -9154.415,E2 -9154.415} C_VEL
LIN {X 0,Y 439.367,Z 346.381,A -85,B 0,C 180,E1 -9157.425,E2 -9157.425} C_VEL
LIN {X 0,Y 439.444,Z 346.37,A -85,B 0,C 180,E1 -9160.663,E2 -9160.663} C_VEL
LIN {X 0,Y 439.466,Z 346.371,A -85,B 0,C 180,E1 -9164.225,E2 -9164.225} C_VEL
LIN {X 0,Y 439.487,Z 346.368,A -85,B 0,C 180,E1 -9168.001,E2 -9168.001} C_VEL
LIN {X 0,Y 439.551,Z 346.359,A -85,B 0,C 180,E1 -9171.726,E2 -9171.726} C_VEL
LIN {X 0,Y 439.624,Z 346.348,A -85,B 0,C 180,E1 -9174.496,E2 -9174.496} C_VEL
LIN {X 0,Y 439.639,Z 346.349,A -85,B 0,C 180,E1 -9178.168,E2 -9178.168} C_VEL
LIN {X 0,Y 439.766,Z 346.331,A -85,B 0,C 180,E1 -9180,E2 -9180} C_VEL
LIN {X 0,Y 439.658,Z 346.345,A -85,B 0,C 180,E1 -9182.749,E2 -9182.749} C_VEL
LIN {X 0,Y 439.622,Z 346.346,A -85,B 0,C 180,E1 -9186.425,E2 -9186.425} C_VEL
LIN {X 0,Y 439.504,Z 346.364,A -85,B 0,C 180,E1 -9189.202,E2 -9189.202} C_VEL
LIN {X 0,Y 439.469,Z 346.349,A -85,B 0,C 180,E1 -9192.938,E2 -9192.938} C_VEL
LIN {X 0,Y 439.451,Z 346.37,A -85,B 0,C 180,E1 -9196.349,E2 -9196.349} C_VEL
LIN {X 0,Y 439.406,Z 346.364,A -85,B 0,C 180,E1 -9199.626,E2 -9199.626} C_VEL
LIN {X 0,Y 439.367,Z 346.378,A -85,B 0,C 180,E1 -9202.575,E2 -9202.575} C_VEL
LIN {X 0,Y 439.401,Z 346.374,A -85,B 0,C 180,E1 -9205.585,E2 -9205.585} C_VEL
LIN {X 0,Y 439.421,Z 346.369,A -85,B 0,C 180,E1 -9208.673,E2 -9208.673} C_VEL
LIN {X 0,Y 439.373,Z 346.376,A -85,B 0,C 180,E1 -9212.03,E2 -9212.03} C_VEL
LIN {X 0,Y 439.399,Z 346.376,A -85,B 0,C 180,E1 -9215.341,E2 -9215.341} C_VEL
LIN {X 0,Y 439.393,Z 346.377,A -85,B 0,C 180,E1 -9218.594,E2 -9218.594} C_VEL
LIN {X 0,Y 439.391,Z 346.38,A -85,B 0,C 180,E1 -9221.257,E2 -9221.257} C_VEL
LIN {X 0,Y 439.404,Z 346.378,A -85,B 0,C 180,E1 -9224.729,E2 -9224.729} C_VEL
LIN {X 0,Y 439.341,Z 346.387,A -85,B 0,C 180,E1 -9227.789,E2 -9227.789} C_VEL
LIN {X 0,Y 439.156,Z 346.41,A -85,B 0,C 180,E1 -9230.198,E2 -9230.198} C_VEL
LIN {X 0,Y 438.993,Z 346.508,A -85,B 0,C 180,E1 -9231.671,E2 -9231.671} C_VEL
LIN {X 0,Y 438.981,Z 349.078,A -85,B 0,C 180,E1 -9234.805,E2 -9234.805} C_VEL
LIN {X 0,Y 438.863,Z 351.875,A -85,B 0,C 180,E1 -9238.098,E2 -9238.098} C_VEL
LIN {X 0,Y 438.773,Z 354.722,A -85,B 0,C 180,E1 -9241.28,E2 -9241.28} C_VEL
LIN {X 0,Y 438.684,Z 357.585,A -85,B 0,C 180,E1 -9244.37,E2 -9244.37} C_VEL
LIN {X 0,Y 438.619,Z 360.035,A -85,B 0,C 180,E1 -9246.797,E2 -9246.797} C_VEL
LIN {X 0,Y 441.959,Z 369.882,A -85,B 0,C 180,E1 -9247.207,E2 -9247.207} C_VEL
LIN {X 0,Y 446.433,Z 384.277,A -85,B 0,C 180,E1 -9247.917,E2 -9247.917} C_VEL
LIN {X 0,Y 447.349,Z 388.253,A -85,B 0,C 180,E1 -9248.125,E2 -9248.125} C_VEL
LIN {X 0,Y 446.631,Z 402.508,A -85,B 0,C 180,E1 -9248.782,E2 -9248.782} C_VEL
LIN {X 0,Y 445.802,Z 416.063,A -85,B 0,C 180,E1 -9249.586,E2 -9249.586} C_VEL
LIN {X 0,Y 444.763,Z 430.037,A -85,B 0,C 180,E1 -9250.619,E2 -9250.619} C_VEL
LIN {X 0,Y 443.726,Z 442.401,A -85,B 0,C 180,E1 -9251.74,E2 -9251.74} C_VEL
LIN {X 0,Y 442.721,Z 453.32,A -85,B 0,C 180,E1 -9252.921,E2 -9252.921} C_VEL
LIN {X 0,Y 441.755,Z 464.09,A -85,B 0,C 180,E1 -9254.308,E2 -9254.308} C_VEL
LIN {X 0,Y 440.956,Z 473.217,A -85,B 0,C 180,E1 -9255.697,E2 -9255.697} C_VEL
LIN {X 0,Y 440.198,Z 482.132,A -85,B 0,C 180,E1 -9257.318,E2 -9257.318} C_VEL
LIN {X 0,Y 439.533,Z 489.52,A -85,B 0,C 180,E1 -9258.937,E2 -9258.937} C_VEL
LIN {X 0,Y 439.087,Z 496.417,A -85,B 0,C 180,E1 -9260.789,E2 -9260.789} C_VEL
LIN {X 0,Y 438.994,Z 497.868,A -85,B 0,C 180,E1 -9261.242,E2 -9261.242} C_VEL
LIN {X 0,Y 438.211,Z 500.078,A -85,B 0,C 180,E1 -9261.95,E2 -9261.95} C_VEL
LIN {X 0,Y 435.166,Z 503.323,A -85,B 0,C 180,E1 -9263.112,E2 -9263.112} C_VEL
LIN {X 0,Y 432.613,Z 505.583,A -85,B 0,C 180,E1 -9264.066,E2 -9264.066} C_VEL
LIN {X 0,Y 431.407,Z 507.273,A -85,B 0,C 180,E1 -9264.942,E2 -9264.942} C_VEL
LIN {X 0,Y 431.371,Z 507.425,A -85,B 0,C 180,E1 -9265.07,E2 -9265.07} C_VEL
LIN {X 0,Y 431.399,Z 509.145,A -85,B 0,C 180,E1 -9266.263,E2 -9266.263} C_VEL
LIN {X 0,Y 431.29,Z 510.876,A -85,B 0,C 180,E1 -9268.132,E2 -9268.132} C_VEL
LIN {X 0,Y 431.23,Z 511.483,A -85,B 0,C 180,E1 -9270,E2 -9270} C_VEL
LIN {X 0,Y 431.29,Z 510.925,A -85,B 0,C 180,E1 -9271.867,E2 -9271.867} C_VEL
LIN {X 0,Y 431.398,Z 509.259,A -85,B 0,C 180,E1 -9273.736,E2 -9273.736} C_VEL
LIN {X 0,Y 431.476,Z 506.45,A -85,B 0,C 180,E1 -9275.608,E2 -9275.608} C_VEL
LIN {X 0,Y 431.702,Z 502.423,A -85,B 0,C 180,E1 -9277.483,E2 -9277.483} C_VEL
LIN {X 0,Y 432.064,Z 497.079,A -85,B 0,C 180,E1 -9279.361,E2 -9279.361} C_VEL
LIN {X 0,Y 432.521,Z 490.269,A -85,B 0,C 180,E1 -9281.244,E2 -9281.244} C_VEL
LIN {X 0,Y 433.208,Z 482.933,A -85,B 0,C 180,E1 -9282.889,E2 -9282.889} C_VEL
LIN {X 0,Y 433.964,Z 474.094,A -85,B 0,C 180,E1 -9284.537,E2 -9284.537} C_VEL
LIN {X 0,Y 434.86,Z 465.07,A -85,B 0,C 180,E1 -9285.946,E2 -9285.946} C_VEL
LIN {X 0,Y 435.843,Z 454.421,A -85,B 0,C 180,E1 -9287.356,E2 -9287.356} C_VEL
LIN {X 0,Y 436.977,Z 442.898,A -85,B 0,C 180,E1 -9288.629,E2 -9288.629} C_VEL
LIN {X 0,Y 438.122,Z 430.065,A -85,B 0,C 180,E1 -9289.808,E2 -9289.808} C_VEL
LIN {X 0,Y 439.198,Z 416.022,A -85,B 0,C 180,E1 -9290.857,E2 -9290.857} C_VEL
LIN {X 0,Y 440.168,Z 401.861,A -85,B 0,C 180,E1 -9291.694,E2 -9291.694} C_VEL
LIN {X 0,Y 440.62,Z 388.753,A -85,B 0,C 180,E1 -9292.314,E2 -9292.314} C_VEL
LIN {X 0,Y 436.362,Z 374.333,A -85,B 0,C 180,E1 -9293.083,E2 -9293.083} C_VEL
LIN {X 0,Y 431.592,Z 360.324,A -85,B 0,C 180,E1 -9293.704,E2 -9293.704} C_VEL
LIN {X 0,Y 431.645,Z 357.054,A -85,B 0,C 180,E1 -9297.122,E2 -9297.122} C_VEL
LIN {X 0,Y 431.738,Z 355.129,A -85,B 0,C 180,E1 -9299.232,E2 -9299.232} C_VEL
LIN {X 0,Y 431.805,Z 352.267,A -85,B 0,C 180,E1 -9302.486,E2 -9302.486} C_VEL
LIN {X 0,Y 431.902,Z 349.71,A -85,B 0,C 180,E1 -9305.55,E2 -9305.55} C_VEL
LIN {X 0,Y 431.978,Z 347.306,A -85,B 0,C 180,E1 -9308.654,E2 -9308.654} C_VEL
LIN {X 0,Y 432.275,Z 347.262,A -85,B 0,C 180,E1 -9311.803,E2 -9311.803} C_VEL
LIN {X 0,Y 432.339,Z 347.256,A -85,B 0,C 180,E1 -9314.346,E2 -9314.346} C_VEL
LIN {X 0,Y 432.319,Z 347.258,A -85,B 0,C 180,E1 -9317.015,E2 -9317.015} C_VEL
LIN {X 0,Y 432.34,Z 347.256,A -85,B 0,C 180,E1 -9319.819,E2 -9319.819} C_VEL
LIN {X 0,Y 432.314,Z 347.258,A -85,B 0,C 180,E1 -9323.023,E2 -9323.023} C_VEL
LIN {X 0,Y 432.358,Z 347.249,A -85,B 0,C 180,E1 -9325.996,E2 -9325.996} C_VEL
LIN {X 0,Y 432.394,Z 347.252,A -85,B 0,C 180,E1 -9329.744,E2 -9329.744} C_VEL
LIN {X 0,Y 432.398,Z 347.24,A -85,B 0,C 180,E1 -9333.372,E2 -9333.372} C_VEL
LIN {X 0,Y 432.37,Z 347.254,A -85,B 0,C 180,E1 -9336.023,E2 -9336.023} C_VEL
LIN {X 0,Y 432.348,Z 347.242,A -85,B 0,C 180,E1 -9339.046,E2 -9339.046} C_VEL
LIN {X 0,Y 432.377,Z 347.251,A -85,B 0,C 180,E1 -9342.011,E2 -9342.011} C_VEL
LIN {X 0,Y 432.394,Z 347.246,A -85,B 0,C 180,E1 -9344.926,E2 -9344.926} C_VEL
LIN {X 0,Y 432.479,Z 347.226,A -85,B 0,C 180,E1 -9347.804,E2 -9347.804} C_VEL
LIN {X 0,Y 432.49,Z 347.236,A -85,B 0,C 180,E1 -9351.59,E2 -9351.59} C_VEL
LIN {X 0,Y 432.596,Z 347.226,A -85,B 0,C 180,E1 -9354.406,E2 -9354.406} C_VEL
LIN {X 0,Y 432.604,Z 347.223,A -85,B 0,C 180,E1 -9358.138,E2 -9358.138} C_VEL
LIN {X 0,Y 432.732,Z 347.21,A -85,B 0,C 180,E1 -9360,E2 -9360} C_VEL
LIN {X 0,Y 432.604,Z 347.223,A -85,B 0,C 180,E1 -9362.793,E2 -9362.793} C_VEL
LIN {X 0,Y 432.571,Z 347.229,A -85,B 0,C 180,E1 -9366.53,E2 -9366.53} C_VEL
LIN {X 0,Y 432.441,Z 347.246,A -85,B 0,C 180,E1 -9369.353,E2 -9369.353} C_VEL
LIN {X 0,Y 432.428,Z 347.244,A -85,B 0,C 180,E1 -9372.804,E2 -9372.804} C_VEL
LIN {X 0,Y 432.41,Z 347.246,A -85,B 0,C 180,E1 -9376.479,E2 -9376.479} C_VEL
LIN {X 0,Y 432.337,Z 347.259,A -85,B 0,C 180,E1 -9379.96,E2 -9379.96} C_VEL
LIN {X 0,Y 432.317,Z 347.262,A -85,B 0,C 180,E1 -9382.964,E2 -9382.964} C_VEL
LIN {X 0,Y 432.362,Z 347.258,A -85,B 0,C 180,E1 -9386.032,E2 -9386.032} C_VEL
LIN {X 0,Y 432.35,Z 347.258,A -85,B 0,C 180,E1 -9389.187,E2 -9389.187} C_VEL
LIN {X 0,Y 432.329,Z 347.259,A -85,B 0,C 180,E1 -9392.295,E2 -9392.295} C_VEL
LIN {X 0,Y 432.339,Z 347.258,A -85,B 0,C 180,E1 -9394.677,E2 -9394.677} C_VEL
LIN {X 0,Y 432.345,Z 347.257,A -85,B 0,C 180,E1 -9398.149,E2 -9398.149} C_VEL
LIN {X 0,Y 432.367,Z 347.417,A -85,B 0,C 180,E1 -9400.863,E2 -9400.863} C_VEL
LIN {X 0,Y 433.282,Z 352.61,A -85,B 0,C 180,E1 -9404.225,E2 -9404.225} C_VEL
LIN {X 0,Y 434.04,Z 357.454,A -85,B 0,C 180,E1 -9407.152,E2 -9407.152} C_VEL
LIN {X 0,Y 434.199,Z 361.769,A -85,B 0,C 180,E1 -9409.53,E2 -9409.53} C_VEL
LIN {X 0,Y 433.654,Z 368.835,A -85,B 0,C 180,E1 -9413.156,E2 -9413.156} C_VEL
LIN {X 0,Y 433.239,Z 375.719,A -85,B 0,C 180,E1 -9416.527,E2 -9416.527} C_VEL
LIN {X 0,Y 432.822,Z 382.61,A -85,B 0,C 180,E1 -9419.778,E2 -9419.778} C_VEL
LIN {X 0,Y 432.414,Z 389.436,A -85,B 0,C 180,E1 -9422.93,E2 -9422.93} C_VEL
LIN {X 0,Y 432.074,Z 396.641,A -85,B 0,C 180,E1 -9426.246,E2 -9426.246} C_VEL
LIN {X 0,Y 432.05,Z 396.805,A -85,B 0,C 180,E1 -9426.32,E2 -9426.32} C_VEL
LIN {X 0,Y 436.548,Z 414.778,A -85,B 0,C 180,E1 -9427.004,E2 -9427.004} C_VEL
LIN {X 0,Y 439.418,Z 429.572,A -85,B 0,C 180,E1 -9427.704,E2 -9427.704} C_VEL
LIN {X 0,Y 439.879,Z 433.776,A -85,B 0,C 180,E1 -9427.922,E2 -9427.922} C_VEL
LIN {X 0,Y 439.056,Z 447.987,A -85,B 0,C 180,E1 -9428.645,E2 -9428.645} C_VEL
LIN {X 0,Y 437.872,Z 462.333,A -85,B 0,C 180,E1 -9429.568,E2 -9429.568} C_VEL
LIN {X 0,Y 436.773,Z 475.409,A -85,B 0,C 180,E1 -9430.618,E2 -9430.618} C_VEL
LIN {X 0,Y 435.674,Z 487.489,A -85,B 0,C 180,E1 -9431.788,E2 -9431.788} C_VEL
LIN {X 0,Y 434.714,Z 498.691,A -85,B 0,C 180,E1 -9433.082,E2 -9433.082} C_VEL
LIN {X 0,Y 433.684,Z 508.997,A -85,B 0,C 180,E1 -9434.492,E2 -9434.492} C_VEL
LIN {X 0,Y 432.839,Z 519.088,A -85,B 0,C 180,E1 -9436.144,E2 -9436.144} C_VEL
LIN {X 0,Y 432.189,Z 528.572,A -85,B 0,C 180,E1 -9438.034,E2 -9438.034} C_VEL
LIN {X 0,Y 431.716,Z 535.363,A -85,B 0,C 180,E1 -9439.685,E2 -9439.685} C_VEL
LIN {X 0,Y 431.456,Z 541.647,A -85,B 0,C 180,E1 -9441.57,E2 -9441.57} C_VEL
LIN {X 0,Y 431.321,Z 546.51,A -85,B 0,C 180,E1 -9443.451,E2 -9443.451} C_VEL
LIN {X 0,Y 431.226,Z 550.074,A -85,B 0,C 180,E1 -9445.326,E2 -9445.326} C_VEL
LIN {X 0,Y 431.259,Z 552.422,A -85,B 0,C 180,E1 -9447.198,E2 -9447.198} C_VEL
LIN {X 0,Y 431.216,Z 553.601,A -85,B 0,C 180,E1 -9449.067,E2 -9449.067} C_VEL
LIN {X 0,Y 431.216,Z 553.6,A -85,B 0,C 180,E1 -9450.934,E2 -9450.934} C_VEL
LIN {X 0,Y 431.259,Z 552.417,A -85,B 0,C 180,E1 -9452.803,E2 -9452.803} C_VEL
LIN {X 0,Y 431.234,Z 550.066,A -85,B 0,C 180,E1 -9454.674,E2 -9454.674} C_VEL
LIN {X 0,Y 431.337,Z 546.507,A -85,B 0,C 180,E1 -9456.549,E2 -9456.549} C_VEL
LIN {X 0,Y 431.457,Z 541.643,A -85,B 0,C 180,E1 -9458.43,E2 -9458.43} C_VEL
LIN {X 0,Y 431.717,Z 535.35,A -85,B 0,C 180,E1 -9460.316,E2 -9460.316} C_VEL
LIN {X 0,Y 432.2,Z 528.555,A -85,B 0,C 180,E1 -9461.966,E2 -9461.966} C_VEL
LIN {X 0,Y 432.841,Z 519.07,A -85,B 0,C 180,E1 -9463.857,E2 -9463.857} C_VEL
LIN {X 0,Y 433.697,Z 508.977,A -85,B 0,C 180,E1 -9465.509,E2 -9465.509} C_VEL
LIN {X 0,Y 434.68,Z 498.666,A -85,B 0,C 180,E1 -9466.92,E2 -9466.92} C_VEL
LIN {X 0,Y 435.743,Z 486.385,A -85,B 0,C 180,E1 -9468.332,E2 -9468.332} C_VEL
LIN {X 0,Y 436.979,Z 472.731,A -85,B 0,C 180,E1 -9469.618,E2 -9469.618} C_VEL
LIN {X 0,Y 438.148,Z 459.051,A -85,B 0,C 180,E1 -9470.664,E2 -9470.664} C_VEL
LIN {X 0,Y 439.216,Z 444.892,A -85,B 0,C 180,E1 -9471.533,E2 -9471.533} C_VEL
LIN {X 0,Y 439.941,Z 432.433,A -85,B 0,C 180,E1 -9472.136,E2 -9472.136} C_VEL
LIN {X 0,Y 437.065,Z 417.206,A -85,B 0,C 180,E1 -9472.883,E2 -9472.883} C_VEL
LIN {X 0,Y 433.418,Z 402.301,A -85,B 0,C 180,E1 -9473.48,E2 -9473.48} C_VEL
LIN {X 0,Y 432.04,Z 396.79,A -85,B 0,C 180,E1 -9473.682,E2 -9473.682} C_VEL
LIN {X 0,Y 432.377,Z 390.397,A -85,B 0,C 180,E1 -9476.621,E2 -9476.621} C_VEL
LIN {X 0,Y 432.745,Z 383.7,A -85,B 0,C 180,E1 -9479.692,E2 -9479.692} C_VEL
LIN {X 0,Y 433.232,Z 375.665,A -85,B 0,C 180,E1 -9483.474,E2 -9483.474} C_VEL
LIN {X 0,Y 433.641,Z 368.754,A -85,B 0,C 180,E1 -9486.846,E2 -9486.846} C_VEL
LIN {X 0,Y 434.123,Z 361.741,A -85,B 0,C 180,E1 -9490.458,E2 -9490.458} C_VEL
LIN {X 0,Y 434.189,Z 359.134,A -85,B 0,C 180,E1 -9491.877,E2 -9491.877} C_VEL
LIN {X 0,Y 433.626,Z 354.605,A -85,B 0,C 180,E1 -9494.51,E2 -9494.51} C_VEL
LIN {X 0,Y 432.927,Z 350.586,A -85,B 0,C 180,E1 -9497.014,E2 -9497.014} C_VEL
LIN {X 0,Y 432.355,Z 347.255,A -85,B 0,C 180,E1 -9499.306,E2 -9499.306} C_VEL
LIN {X 0,Y 432.349,Z 347.259,A -85,B 0,C 180,E1 -9501.851,E2 -9501.851} C_VEL
LIN {X 0,Y 432.343,Z 347.259,A -85,B 0,C 180,E1 -9505.323,E2 -9505.323} C_VEL
LIN {X 0,Y 432.323,Z 347.259,A -85,B 0,C 180,E1 -9508.654,E2 -9508.654} C_VEL
LIN {X 0,Y 432.385,Z 347.251,A -85,B 0,C 180,E1 -9511.877,E2 -9511.877} C_VEL
LIN {X 0,Y 432.351,Z 347.256,A -85,B 0,C 180,E1 -9514.999,E2 -9514.999} C_VEL
LIN {X 0,Y 432.36,Z 347.254,A -85,B 0,C 180,E1 -9518.046,E2 -9518.046} C_VEL
LIN {X 0,Y 432.39,Z 347.25,A -85,B 0,C 180,E1 -9521.03,E2 -9521.03} C_VEL
LIN {X 0,Y 432.434,Z 347.245,A -85,B 0,C 180,E1 -9523.961,E2 -9523.961} C_VEL
LIN {X 0,Y 432.462,Z 347.245,A -85,B 0,C 180,E1 -9527.804,E2 -9527.804} C_VEL
LIN {X 0,Y 432.495,Z 347.237,A -85,B 0,C 180,E1 -9531.59,E2 -9531.59} C_VEL
LIN {X 0,Y 432.601,Z 347.223,A -85,B 0,C 180,E1 -9534.406,E2 -9534.406} C_VEL
LIN {X 0,Y 432.609,Z 347.224,A -85,B 0,C 180,E1 -9538.138,E2 -9538.138} C_VEL
LIN {X 0,Y 432.735,Z 347.207,A -85,B 0,C 180,E1 -9540,E2 -9540} C_VEL
LIN {X 0,Y 432.608,Z 347.223,A -85,B 0,C 180,E1 -9542.794,E2 -9542.794} C_VEL
LIN {X 0,Y 432.577,Z 347.223,A -85,B 0,C 180,E1 -9546.53,E2 -9546.53} C_VEL
LIN {X 0,Y 432.447,Z 347.242,A -85,B 0,C 180,E1 -9549.353,E2 -9549.353} C_VEL
LIN {X 0,Y 432.434,Z 347.225,A -85,B 0,C 180,E1 -9552.803,E2 -9552.803} C_VEL
LIN {X 0,Y 432.416,Z 347.248,A -85,B 0,C 180,E1 -9556.479,E2 -9556.479} C_VEL
LIN {X 0,Y 432.342,Z 347.24,A -85,B 0,C 180,E1 -9559.96,E2 -9559.96} C_VEL
LIN {X 0,Y 432.321,Z 347.258,A -85,B 0,C 180,E1 -9562.964,E2 -9562.964} C_VEL
LIN {X 0,Y 432.364,Z 347.245,A -85,B 0,C 180,E1 -9566.033,E2 -9566.033} C_VEL
LIN {X 0,Y 432.346,Z 347.254,A -85,B 0,C 180,E1 -9569.187,E2 -9569.187} C_VEL
LIN {X 0,Y 432.326,Z 347.251,A -85,B 0,C 180,E1 -9572.443,E2 -9572.443} C_VEL
LIN {X 0,Y 432.349,Z 347.254,A -85,B 0,C 180,E1 -9575.632,E2 -9575.632} C_VEL
LIN {X 0,Y 432.356,Z 347.254,A -85,B 0,C 180,E1 -9578.716,E2 -9578.716} C_VEL
LIN {X 0,Y 432.336,Z 347.257,A -85,B 0,C 180,E1 -9581.797,E2 -9581.797} C_VEL
LIN {X 0,Y 432.336,Z 347.26,A -85,B 0,C 180,E1 -9584.347,E2 -9584.347} C_VEL
LIN {X 0,Y 432.312,Z 347.265,A -85,B 0,C 180,E1 -9587.017,E2 -9587.017} C_VEL
LIN {X 0,Y 432.143,Z 347.284,A -85,B 0,C 180,E1 -9589.851,E2 -9589.851} C_VEL
LIN {X 0,Y 431.935,Z 347.462,A -85,B 0,C 180,E1 -9591.808,E2 -9591.808} C_VEL
LIN {X 0,Y 431.893,Z 350.308,A -85,B 0,C 180,E1 -9595.282,E2 -9595.282} C_VEL
LIN {X 0,Y 431.794,Z 353.104,A -85,B 0,C 180,E1 -9598.611,E2 -9598.611} C_VEL
LIN {X 0,Y 431.739,Z 355.986,A -85,B 0,C 180,E1 -9601.831,E2 -9601.831} C_VEL
LIN {X 0,Y 431.622,Z 358.93,A -85,B 0,C 180,E1 -9604.953,E2 -9604.953} C_VEL
LIN {X 0,Y 431.611,Z 360.504,A -85,B 0,C 180,E1 -9606.399,E2 -9606.399} C_VEL
LIN {X 0,Y 435.056,Z 370.578,A -85,B 0,C 180,E1 -9606.833,E2 -9606.833} C_VEL
LIN {X 0,Y 439.66,Z 385.099,A -85,B 0,C 180,E1 -9607.576,E2 -9607.576} C_VEL
LIN {X 0,Y 440.742,Z 389.235,A -85,B 0,C 180,E1 -9607.805,E2 -9607.805} C_VEL
LIN {X 0,Y 439.977,Z 403.986,A -85,B 0,C 180,E1 -9608.506,E2 -9608.506} C_VEL
LIN {X 0,Y 439.035,Z 418.173,A -85,B 0,C 180,E1 -9609.379,E2 -9609.379} C_VEL
LIN {X 0,Y 437.943,Z 431.808,A -85,B 0,C 180,E1 -9610.427,E2 -9610.427} C_VEL
LIN {X 0,Y 436.796,Z 444.568,A -85,B 0,C 180,E1 -9611.629,E2 -9611.629} C_VEL
LIN {X 0,Y 435.771,Z 455.603,A -85,B 0,C 180,E1 -9612.882,E2 -9612.882} C_VEL
LIN {X 0,Y 434.742,Z 466.053,A -85,B 0,C 180,E1 -9614.289,E2 -9614.289} C_VEL
LIN {X 0,Y 433.758,Z 476.246,A -85,B 0,C 180,E1 -9615.934,E2 -9615.934} C_VEL
LIN {X 0,Y 433.098,Z 484.696,A -85,B 0,C 180,E1 -9617.583,E2 -9617.583} C_VEL
LIN {X 0,Y 432.414,Z 491.732,A -85,B 0,C 180,E1 -9619.227,E2 -9619.227} C_VEL
LIN {X 0,Y 431.947,Z 498.468,A -85,B 0,C 180,E1 -9621.182,E2 -9621.182} C_VEL
LIN {X 0,Y 431.629,Z 503.446,A -85,B 0,C 180,E1 -9623.032,E2 -9623.032} C_VEL
LIN {X 0,Y 431.371,Z 507.425,A -85,B 0,C 180,E1 -9625.07,E2 -9625.07} C_VEL
LIN {X 0,Y 430.645,Z 508.671,A -85,B 0,C 180,E1 -9625.832,E2 -9625.832} C_VEL
LIN {X 0,Y 427.747,Z 510.335,A -85,B 0,C 180,E1 -9627.079,E2 -9627.079} C_VEL
LIN {X 0,Y 425.315,Z 511.244,A -85,B 0,C 180,E1 -9628.093,E2 -9628.093} C_VEL
LIN {X 0,Y 424.253,Z 511.627,A -85,B 0,C 180,E1 -9628.88,E2 -9628.88} C_VEL
LIN {X 0,Y 424.155,Z 511.689,A -85,B 0,C 180,E1 -9629.147,E2 -9629.147} C_VEL
LIN {X 0,Y 424.163,Z 511.689,A -85,B 0,C 180,E1 -9630.949,E2 -9630.949} C_VEL
LIN {X 0,Y 424.29,Z 510.578,A -85,B 0,C 180,E1 -9632.848,E2 -9632.848} C_VEL
LIN {X 0,Y 424.273,Z 508.353,A -85,B 0,C 180,E1 -9634.75,E2 -9634.75} C_VEL
LIN {X 0,Y 424.5,Z 504.942,A -85,B 0,C 180,E1 -9636.655,E2 -9636.655} C_VEL
LIN {X 0,Y 424.805,Z 500.272,A -85,B 0,C 180,E1 -9638.563,E2 -9638.563} C_VEL
LIN {X 0,Y 425.266,Z 494.218,A -85,B 0,C 180,E1 -9640.473,E2 -9640.473} C_VEL
LIN {X 0,Y 426.007,Z 486.583,A -85,B 0,C 180,E1 -9642.384,E2 -9642.384} C_VEL
LIN {X 0,Y 426.688,Z 478.572,A -85,B 0,C 180,E1 -9644.036,E2 -9644.036} C_VEL
LIN {X 0,Y 427.693,Z 468.629,A -85,B 0,C 180,E1 -9645.731,E2 -9645.731} C_VEL
LIN {X 0,Y 428.693,Z 458.557,A -85,B 0,C 180,E1 -9647.163,E2 -9647.163} C_VEL
LIN {X 0,Y 429.8,Z 447.484,A -85,B 0,C 180,E1 -9648.485,E2 -9648.485} C_VEL
LIN {X 0,Y 430.884,Z 435.795,A -85,B 0,C 180,E1 -9649.658,E2 -9649.658} C_VEL
LIN {X 0,Y 432.08,Z 422.986,A -85,B 0,C 180,E1 -9650.718,E2 -9650.718} C_VEL
LIN {X 0,Y 433.129,Z 408.933,A -85,B 0,C 180,E1 -9651.662,E2 -9651.662} C_VEL
LIN {X 0,Y 433.986,Z 394.189,A -85,B 0,C 180,E1 -9652.437,E2 -9652.437} C_VEL
LIN {X 0,Y 433.925,Z 389.997,A -85,B 0,C 180,E1 -9652.64,E2 -9652.64} C_VEL
LIN {X 0,Y 429.679,Z 375.645,A -85,B 0,C 180,E1 -9653.434,E2 -9653.434} C_VEL
LIN {X 0,Y 424.655,Z 361.263,A -85,B 0,C 180,E1 -9654.1,E2 -9654.1} C_VEL
LIN {X 0,Y 424.57,Z 360.664,A -85,B 0,C 180,E1 -9654.132,E2 -9654.132} C_VEL
LIN {X 0,Y 424.61,Z 357.382,A -85,B 0,C 180,E1 -9657.609,E2 -9657.609} C_VEL
LIN {X 0,Y 424.718,Z 354.469,A -85,B 0,C 180,E1 -9660.861,E2 -9660.861} C_VEL
LIN {X 0,Y 424.821,Z 351.609,A -85,B 0,C 180,E1 -9664.227,E2 -9664.227} C_VEL
LIN {X 0,Y 424.887,Z 348.761,A -85,B 0,C 180,E1 -9667.735,E2 -9667.735} C_VEL
LIN {X 0,Y 424.963,Z 348.178,A -85,B 0,C 180,E1 -9668.987,E2 -9668.987} C_VEL
LIN {X 0,Y 425.224,Z 348.14,A -85,B 0,C 180,E1 -9671.948,E2 -9671.948} C_VEL
LIN {X 0,Y 425.285,Z 348.134,A -85,B 0,C 180,E1 -9675.282,E2 -9675.282} C_VEL
LIN {X 0,Y 425.274,Z 348.136,A -85,B 0,C 180,E1 -9678.621,E2 -9678.621} C_VEL
LIN {X 0,Y 425.314,Z 348.131,A -85,B 0,C 180,E1 -9681.103,E2 -9681.103} C_VEL
LIN {X 0,Y 425.299,Z 348.133,A -85,B 0,C 180,E1 -9684.664,E2 -9684.664} C_VEL
LIN {X 0,Y 425.266,Z 348.132,A -85,B 0,C 180,E1 -9688.073,E2 -9688.073} C_VEL
LIN {X 0,Y 425.336,Z 348.124,A -85,B 0,C 180,E1 -9691.368,E2 -9691.368} C_VEL
LIN {X 0,Y 425.294,Z 348.132,A -85,B 0,C 180,E1 -9694.554,E2 -9694.554} C_VEL
LIN {X 0,Y 425.286,Z 348.13,A -85,B 0,C 180,E1 -9697.661,E2 -9697.661} C_VEL
LIN {X 0,Y 425.36,Z 348.118,A -85,B 0,C 180,E1 -9700.704,E2 -9700.704} C_VEL
LIN {X 0,Y 425.386,Z 348.122,A -85,B 0,C 180,E1 -9703.688,E2 -9703.688} C_VEL
LIN {X 0,Y 425.428,Z 348.103,A -85,B 0,C 180,E1 -9707.599,E2 -9707.599} C_VEL
LIN {X 0,Y 425.441,Z 348.115,A -85,B 0,C 180,E1 -9711.45,E2 -9711.45} C_VEL
LIN {X 0,Y 425.553,Z 348.104,A -85,B 0,C 180,E1 -9714.313,E2 -9714.313} C_VEL
LIN {X 0,Y 425.574,Z 348.099,A -85,B 0,C 180,E1 -9718.107,E2 -9718.107} C_VEL
LIN {X 0,Y 425.701,Z 348.085,A -85,B 0,C 180,E1 -9720,E2 -9720} C_VEL
LIN {X 0,Y 425.556,Z 348.101,A -85,B 0,C 180,E1 -9722.84,E2 -9722.84} C_VEL
LIN {X 0,Y 425.529,Z 348.106,A -85,B 0,C 180,E1 -9726.639,E2 -9726.639} C_VEL
LIN {X 0,Y 425.4,Z 348.122,A -85,B 0,C 180,E1 -9729.509,E2 -9729.509} C_VEL
LIN {X 0,Y 425.391,Z 348.12,A -85,B 0,C 180,E1 -9732.904,E2 -9732.904} C_VEL
LIN {X 0,Y 425.359,Z 348.125,A -85,B 0,C 180,E1 -9736.605,E2 -9736.605} C_VEL
LIN {X 0,Y 425.326,Z 348.13,A -85,B 0,C 180,E1 -9739.636,E2 -9739.636} C_VEL
LIN {X 0,Y 425.305,Z 348.135,A -85,B 0,C 180,E1 -9743.365,E2 -9743.365} C_VEL
LIN {X 0,Y 425.346,Z 348.129,A -85,B 0,C 180,E1 -9746.845,E2 -9746.845} C_VEL
LIN {X 0,Y 425.316,Z 348.132,A -85,B 0,C 180,E1 -9749.717,E2 -9749.717} C_VEL
LIN {X 0,Y 425.282,Z 348.136,A -85,B 0,C 180,E1 -9753.048,E2 -9753.048} C_VEL
LIN {X 0,Y 425.282,Z 348.137,A -85,B 0,C 180,E1 -9755.929,E2 -9755.929} C_VEL
LIN {X 0,Y 425.301,Z 348.133,A -85,B 0,C 180,E1 -9759.045,E2 -9759.045} C_VEL
LIN {X 0,Y 425.318,Z 348.288,A -85,B 0,C 180,E1 -9760.441,E2 -9760.441} C_VEL
LIN {X 0,Y 426.198,Z 353.378,A -85,B 0,C 180,E1 -9763.834,E2 -9763.834} C_VEL
LIN {X 0,Y 426.885,Z 357.527,A -85,B 0,C 180,E1 -9766.418,E2 -9766.418} C_VEL
LIN {X 0,Y 427.216,Z 361.777,A -85,B 0,C 180,E1 -9768.851,E2 -9768.851} C_VEL
LIN {X 0,Y 426.886,Z 366.317,A -85,B 0,C 180,E1 -9771.274,E2 -9771.274} C_VEL
LIN {X 0,Y 426.57,Z 371.285,A -85,B 0,C 180,E1 -9773.833,E2 -9773.833} C_VEL
LIN {X 0,Y 426.097,Z 378.23,A -85,B 0,C 180,E1 -9777.266,E2 -9777.266} C_VEL
LIN {X 0,Y 425.698,Z 384.59,A -85,B 0,C 180,E1 -9780.312,E2 -9780.312} C_VEL
LIN {X 0,Y 425.248,Z 392.461,A -85,B 0,C 180,E1 -9784.027,E2 -9784.027} C_VEL
LIN {X 0,Y 425.031,Z 396.63,A -85,B 0,C 180,E1 -9785.918,E2 -9785.918} C_VEL
LIN {X 0,Y 429.288,Z 413.304,A -85,B 0,C 180,E1 -9786.56,E2 -9786.56} C_VEL
LIN {X 0,Y 432.142,Z 427.161,A -85,B 0,C 180,E1 -9787.224,E2 -9787.224} C_VEL
LIN {X 0,Y 433.217,Z 434.666,A -85,B 0,C 180,E1 -9787.623,E2 -9787.623} C_VEL
LIN {X 0,Y 432.264,Z 449.639,A -85,B 0,C 180,E1 -9788.417,E2 -9788.417} C_VEL
LIN {X 0,Y 431.034,Z 463.576,A -85,B 0,C 180,E1 -9789.354,E2 -9789.354} C_VEL
LIN {X 0,Y 429.9,Z 476.36,A -85,B 0,C 180,E1 -9790.42,E2 -9790.42} C_VEL
LIN {X 0,Y 428.649,Z 489.296,A -85,B 0,C 180,E1 -9791.726,E2 -9791.726} C_VEL
LIN {X 0,Y 427.659,Z 500.14,A -85,B 0,C 180,E1 -9793.041,E2 -9793.041} C_VEL
LIN {X 0,Y 426.612,Z 510.175,A -85,B 0,C 180,E1 -9794.473,E2 -9794.473} C_VEL
LIN {X 0,Y 425.758,Z 520.007,A -85,B 0,C 180,E1 -9796.152,E2 -9796.152} C_VEL
LIN {X 0,Y 425.182,Z 528.222,A -85,B 0,C 180,E1 -9797.834,E2 -9797.834} C_VEL
LIN {X 0,Y 424.689,Z 535.014,A -85,B 0,C 180,E1 -9799.512,E2 -9799.512} C_VEL
LIN {X 0,Y 424.385,Z 541.297,A -85,B 0,C 180,E1 -9801.429,E2 -9801.429} C_VEL
LIN {X 0,Y 424.23,Z 546.161,A -85,B 0,C 180,E1 -9803.341,E2 -9803.341} C_VEL
LIN {X 0,Y 424.153,Z 549.726,A -85,B 0,C 180,E1 -9805.248,E2 -9805.248} C_VEL
LIN {X 0,Y 424.172,Z 552.075,A -85,B 0,C 180,E1 -9807.151,E2 -9807.151} C_VEL
LIN {X 0,Y 424.132,Z 553.254,A -85,B 0,C 180,E1 -9809.051,E2 -9809.051} C_VEL
LIN {X 0,Y 424.132,Z 553.253,A -85,B 0,C 180,E1 -9810.95,E2 -9810.95} C_VEL
LIN {X 0,Y 424.172,Z 552.069,A -85,B 0,C 180,E1 -9812.85,E2 -9812.85} C_VEL
LIN {X 0,Y 424.162,Z 549.718,A -85,B 0,C 180,E1 -9814.753,E2 -9814.753} C_VEL
LIN {X 0,Y 424.247,Z 546.157,A -85,B 0,C 180,E1 -9816.659,E2 -9816.659} C_VEL
LIN {X 0,Y 424.385,Z 541.292,A -85,B 0,C 180,E1 -9818.572,E2 -9818.572} C_VEL
LIN {X 0,Y 424.69,Z 534.999,A -85,B 0,C 180,E1 -9820.489,E2 -9820.489} C_VEL
LIN {X 0,Y 425.194,Z 528.203,A -85,B 0,C 180,E1 -9822.166,E2 -9822.166} C_VEL
LIN {X 0,Y 425.867,Z 518.717,A -85,B 0,C 180,E1 -9824.089,E2 -9824.089} C_VEL
LIN {X 0,Y 426.77,Z 508.623,A -85,B 0,C 180,E1 -9825.767,E2 -9825.767} C_VEL
LIN {X 0,Y 427.919,Z 497.115,A -85,B 0,C 180,E1 -9827.351,E2 -9827.351} C_VEL
LIN {X 0,Y 429.076,Z 484.877,A -85,B 0,C 180,E1 -9828.751,E2 -9828.751} C_VEL
LIN {X 0,Y 430.244,Z 472.376,A -85,B 0,C 180,E1 -9829.938,E2 -9829.938} C_VEL
LIN {X 0,Y 431.468,Z 458.697,A -85,B 0,C 180,E1 -9830.999,E2 -9830.999} C_VEL
LIN {X 0,Y 432.596,Z 444.538,A -85,B 0,C 180,E1 -9831.879,E2 -9831.879} C_VEL
LIN {X 0,Y 433.164,Z 433.135,A -85,B 0,C 180,E1 -9832.45,E2 -9832.45} C_VEL
LIN {X 0,Y 430.317,Z 417.916,A -85,B 0,C 180,E1 -9833.225,E2 -9833.225} C_VEL
LIN {X 0,Y 426.512,Z 402.267,A -85,B 0,C 180,E1 -9833.876,E2 -9833.876} C_VEL
LIN {X 0,Y 425.029,Z 396.452,A -85,B 0,C 180,E1 -9834.091,E2 -9834.091} C_VEL
LIN {X 0,Y 425.333,Z 390.623,A -85,B 0,C 180,E1 -9836.84,E2 -9836.84} C_VEL
LIN {X 0,Y 425.704,Z 384.531,A -85,B 0,C 180,E1 -9839.688,E2 -9839.688} C_VEL
LIN {X 0,Y 426.212,Z 376.551,A -85,B 0,C 180,E1 -9843.532,E2 -9843.532} C_VEL
LIN {X 0,Y 426.644,Z 369.624,A -85,B 0,C 180,E1 -9846.96,E2 -9846.96} C_VEL
LIN {X 0,Y 427.178,Z 362.307,A -85,B 0,C 180,E1 -9850.817,E2 -9850.817} C_VEL
LIN {X 0,Y 427.113,Z 359.457,A -85,B 0,C 180,E1 -9852.427,E2 -9852.427} C_VEL
LIN {X 0,Y 426.489,Z 354.977,A -85,B 0,C 180,E1 -9855.12,E2 -9855.12} C_VEL
LIN {X 0,Y 425.557,Z 349.55,A -85,B 0,C 180,E1 -9858.655,E2 -9858.655} C_VEL
LIN {X 0,Y 425.313,Z 348.133,A -85,B 0,C 180,E1 -9859.673,E2 -9859.673} C_VEL
LIN {X 0,Y 425.287,Z 348.14,A -85,B 0,C 180,E1 -9862.488,E2 -9862.488} C_VEL
LIN {X 0,Y 425.31,Z 348.135,A -85,B 0,C 180,E1 -9865.818,E2 -9865.818} C_VEL
LIN {X 0,Y 425.293,Z 348.134,A -85,B 0,C 180,E1 -9869.239,E2 -9869.239} C_VEL
LIN {X 0,Y 425.352,Z 348.13,A -85,B 0,C 180,E1 -9872.443,E2 -9872.443} C_VEL
LIN {X 0,Y 425.352,Z 348.129,A -85,B 0,C 180,E1 -9875.602,E2 -9875.602} C_VEL
LIN {X 0,Y 425.296,Z 348.136,A -85,B 0,C 180,E1 -9878.682,E2 -9878.682} C_VEL
LIN {X 0,Y 425.336,Z 348.131,A -85,B 0,C 180,E1 -9881.703,E2 -9881.703} C_VEL
LIN {X 0,Y 425.352,Z 348.131,A -85,B 0,C 180,E1 -9884.671,E2 -9884.671} C_VEL
LIN {X 0,Y 425.415,Z 348.124,A -85,B 0,C 180,E1 -9887.598,E2 -9887.598} C_VEL
LIN {X 0,Y 425.446,Z 348.115,A -85,B 0,C 180,E1 -9891.45,E2 -9891.45} C_VEL
LIN {X 0,Y 425.557,Z 348.101,A -85,B 0,C 180,E1 -9894.313,E2 -9894.313} C_VEL
LIN {X 0,Y 425.579,Z 348.1,A -85,B 0,C 180,E1 -9898.107,E2 -9898.107} C_VEL
LIN {X 0,Y 425.705,Z 348.083,A -85,B 0,C 180,E1 -9900,E2 -9900} C_VEL
LIN {X 0,Y 425.559,Z 348.1,A -85,B 0,C 180,E1 -9902.84,E2 -9902.84} C_VEL
LIN {X 0,Y 425.535,Z 348.1,A -85,B 0,C 180,E1 -9906.639,E2 -9906.639} C_VEL
LIN {X 0,Y 425.405,Z 348.119,A -85,B 0,C 180,E1 -9909.509,E2 -9909.509} C_VEL
LIN {X 0,Y 425.397,Z 348.101,A -85,B 0,C 180,E1 -9912.904,E2 -9912.904} C_VEL
LIN {X 0,Y 425.365,Z 348.127,A -85,B 0,C 180,E1 -9916.605,E2 -9916.605} C_VEL
LIN {X 0,Y 425.332,Z 348.115,A -85,B 0,C 180,E1 -9919.636,E2 -9919.636} C_VEL
LIN {X 0,Y 425.291,Z 348.129,A -85,B 0,C 180,E1 -9922.339,E2 -9922.339} C_VEL
LIN {X 0,Y 425.294,Z 348.133,A -85,B 0,C 180,E1 -9925.446,E2 -9925.446} C_VEL
LIN {X 0,Y 425.351,Z 348.116,A -85,B 0,C 180,E1 -9927.558,E2 -9927.558} C_VEL
LIN {X 0,Y 425.291,Z 348.133,A -85,B 0,C 180,E1 -9930.816,E2 -9930.816} C_VEL
LIN {X 0,Y 425.315,Z 348.124,A -85,B 0,C 180,E1 -9934.288,E2 -9934.288} C_VEL
LIN {X 0,Y 425.289,Z 348.136,A -85,B 0,C 180,E1 -9937.693,E2 -9937.693} C_VEL
LIN {X 0,Y 425.287,Z 348.136,A -85,B 0,C 180,E1 -9940.521,E2 -9940.521} C_VEL
LIN {X 0,Y 425.26,Z 348.139,A -85,B 0,C 180,E1 -9943.351,E2 -9943.351} C_VEL
LIN {X 0,Y 425.267,Z 348.14,A -85,B 0,C 180,E1 -9946.044,E2 -9946.044} C_VEL
LIN {X 0,Y 425.201,Z 348.151,A -85,B 0,C 180,E1 -9948.612,E2 -9948.612} C_VEL
LIN {X 0,Y 424.974,Z 348.177,A -85,B 0,C 180,E1 -9951.066,E2 -9951.066} C_VEL
LIN {X 0,Y 424.886,Z 348.904,A -85,B 0,C 180,E1 -9952.558,E2 -9952.558} C_VEL
LIN {X 0,Y 424.826,Z 351.54,A -85,B 0,C 180,E1 -9955.808,E2 -9955.808} C_VEL
LIN {X 0,Y 424.73,Z 354.581,A -85,B 0,C 180,E1 -9959.366,E2 -9959.366} C_VEL
LIN {X 0,Y 424.632,Z 357.284,A -85,B 0,C 180,E1 -9962.391,E2 -9962.391} C_VEL
LIN {X 0,Y 424.567,Z 360.703,A -85,B 0,C 180,E1 -9965.963,E2 -9965.963} C_VEL
LIN {X 0,Y 430.602,Z 378.536,A -85,B 0,C 180,E1 -9966.815,E2 -9966.815} C_VEL
LIN {X 0,Y 433.821,Z 389.585,A -85,B 0,C 180,E1 -9967.431,E2 -9967.431} C_VEL
LIN {X 0,Y 434.087,Z 392.682,A -85,B 0,C 180,E1 -9967.589,E2 -9967.589} C_VEL
LIN {X 0,Y 433.228,Z 407.424,A -85,B 0,C 180,E1 -9968.342,E2 -9968.342} C_VEL
LIN {X 0,Y 432.289,Z 420.208,A -85,B 0,C 180,E1 -9969.167,E2 -9969.167} C_VEL
LIN {X 0,Y 431.156,Z 433.534,A -85,B 0,C 180,E1 -9970.23,E2 -9970.23} C_VEL
LIN {X 0,Y 429.969,Z 446.039,A -85,B 0,C 180,E1 -9971.448,E2 -9971.448} C_VEL
LIN {X 0,Y 428.8,Z 457.872,A -85,B 0,C 180,E1 -9972.841,E2 -9972.841} C_VEL
LIN {X 0,Y 427.764,Z 468.014,A -85,B 0,C 180,E1 -9974.271,E2 -9974.271} C_VEL
LIN {X 0,Y 426.744,Z 478.067,A -85,B 0,C 180,E1 -9975.965,E2 -9975.965} C_VEL
LIN {X 0,Y 426.083,Z 486.146,A -85,B 0,C 180,E1 -9977.618,E2 -9977.618} C_VEL
LIN {X 0,Y 425.423,Z 492.083,A -85,B 0,C 180,E1 -9979.048,E2 -9979.048} C_VEL
LIN {X 0,Y 424.952,Z 498.598,A -85,B 0,C 180,E1 -9980.96,E2 -9980.96} C_VEL
LIN {X 0,Y 424.581,Z 503.691,A -85,B 0,C 180,E1 -9982.868,E2 -9982.868} C_VEL
LIN {X 0,Y 424.427,Z 506.622,A -85,B 0,C 180,E1 -9984.298,E2 -9984.298} C_VEL
LIN {X 0,Y 424.306,Z 509.494,A -85,B 0,C 180,E1 -9986.201,E2 -9986.201} C_VEL
LIN {X 0,Y 424.213,Z 511.223,A -85,B 0,C 180,E1 -9988.101,E2 -9988.101} C_VEL
LIN {X 0,Y 424.155,Z 511.689,A -85,B 0,C 180,E1 -9989.147,E2 -9989.147} C_VEL
LIN {X 0,Y 423.47,Z 511.854,A -85,B 0,C 180,E1 -9989.94,E2 -9989.94} C_VEL
LIN {X 0,Y 420.658,Z 511.781,A -85,B 0,C 180,E1 -9991.231,E2 -9991.231} C_VEL
LIN {X 0,Y 418.299,Z 511.374,A -85,B 0,C 180,E1 -9992.27,E2 -9992.27} C_VEL
LIN {X 0,Y 417.287,Z 510.781,A -85,B 0,C 180,E1 -9993.069,E2 -9993.069} C_VEL
LIN {X 0,Y 417.204,Z 510.48,A -85,B 0,C 180,E1 -9993.339,E2 -9993.339} C_VEL
LIN {X 0,Y 417.207,Z 508.7,A -85,B 0,C 180,E1 -9994.831,E2 -9994.831} C_VEL
LIN {X 0,Y 417.442,Z 505.289,A -85,B 0,C 180,E1 -9996.768,E2 -9996.768} C_VEL
LIN {X 0,Y 417.78,Z 500.619,A -85,B 0,C 180,E1 -9998.708,E2 -9998.708} C_VEL
LIN {X 0,Y 418.268,Z 494.565,A -85,B 0,C 180,E1 -10000.651,E2 -10000.651} C_VEL
LIN {X 0,Y 419.026,Z 486.932,A -85,B 0,C 180,E1 -10002.593,E2 -10002.593} C_VEL
LIN {X 0,Y 419.77,Z 478.919,A -85,B 0,C 180,E1 -10004.272,E2 -10004.272} C_VEL
LIN {X 0,Y 420.831,Z 468.975,A -85,B 0,C 180,E1 -10005.995,E2 -10005.995} C_VEL
LIN {X 0,Y 421.886,Z 458.903,A -85,B 0,C 180,E1 -10007.448,E2 -10007.448} C_VEL
LIN {X 0,Y 423.171,Z 446.995,A -85,B 0,C 180,E1 -10008.884,E2 -10008.884} C_VEL
LIN {X 0,Y 424.379,Z 434.854,A -85,B 0,C 180,E1 -10010.098,E2 -10010.098} C_VEL
LIN {X 0,Y 425.526,Z 421.76,A -85,B 0,C 180,E1 -10011.179,E2 -10011.179} C_VEL
LIN {X 0,Y 426.56,Z 409.273,A -85,B 0,C 180,E1 -10012.013,E2 -10012.013} C_VEL
LIN {X 0,Y 427.406,Z 395.236,A -85,B 0,C 180,E1 -10012.767,E2 -10012.767} C_VEL
LIN {X 0,Y 427.376,Z 391.715,A -85,B 0,C 180,E1 -10012.943,E2 -10012.943} C_VEL
LIN {X 0,Y 423.274,Z 377.741,A -85,B 0,C 180,E1 -10013.749,E2 -10013.749} C_VEL
LIN {X 0,Y 418.254,Z 363.563,A -85,B 0,C 180,E1 -10014.449,E2 -10014.449} C_VEL
LIN {X 0,Y 417.525,Z 361.008,A -85,B 0,C 180,E1 -10014.574,E2 -10014.574} C_VEL
LIN {X 0,Y 417.566,Z 357.719,A -85,B 0,C 180,E1 -10018.116,E2 -10018.116} C_VEL
LIN {X 0,Y 417.667,Z 354.781,A -85,B 0,C 180,E1 -10021.441,E2 -10021.441} C_VEL
LIN {X 0,Y 417.786,Z 351.901,A -85,B 0,C 180,E1 -10024.886,E2 -10024.886} C_VEL
LIN {X 0,Y 417.864,Z 349.064,A -85,B 0,C 180,E1 -10028.484,E2 -10028.484} C_VEL
LIN {X 0,Y 418.126,Z 349.026,A -85,B 0,C 180,E1 -10030.959,E2 -10030.959} C_VEL
LIN {X 0,Y 418.209,Z 349.014,A -85,B 0,C 180,E1 -10033.729,E2 -10033.729} C_VEL
LIN {X 0,Y 418.208,Z 349.017,A -85,B 0,C 180,E1 -10036.448,E2 -10036.448} C_VEL
LIN {X 0,Y 418.223,Z 349.017,A -85,B 0,C 180,E1 -10039.13,E2 -10039.13} C_VEL
LIN {X 0,Y 418.234,Z 349.016,A -85,B 0,C 180,E1 -10042.165,E2 -10042.165} C_VEL
LIN {X 0,Y 418.264,Z 349.007,A -85,B 0,C 180,E1 -10045.419,E2 -10045.419} C_VEL
LIN {X 0,Y 418.217,Z 349.015,A -85,B 0,C 180,E1 -10048.604,E2 -10048.604} C_VEL
LIN {X 0,Y 418.294,Z 348.998,A -85,B 0,C 180,E1 -10051.937,E2 -10051.937} C_VEL
LIN {X 0,Y 418.288,Z 349.004,A -85,B 0,C 180,E1 -10055.162,E2 -10055.162} C_VEL
LIN {X 0,Y 418.232,Z 349.007,A -85,B 0,C 180,E1 -10058.303,E2 -10058.303} C_VEL
LIN {X 0,Y 418.282,Z 349.001,A -85,B 0,C 180,E1 -10061.383,E2 -10061.383} C_VEL
LIN {X 0,Y 418.3,Z 349.002,A -85,B 0,C 180,E1 -10064.406,E2 -10064.406} C_VEL
LIN {X 0,Y 418.368,Z 348.981,A -85,B 0,C 180,E1 -10067.386,E2 -10067.386} C_VEL
LIN {X 0,Y 418.358,Z 348.997,A -85,B 0,C 180,E1 -10070.329,E2 -10070.329} C_VEL
LIN {X 0,Y 418.492,Z 348.98,A -85,B 0,C 180,E1 -10073.249,E2 -10073.249} C_VEL
LIN {X 0,Y 418.339,Z 349,A -85,B 0,C 180,E1 -10075.181,E2 -10075.181} C_VEL
LIN {X 0,Y 418.543,Z 348.974,A -85,B 0,C 180,E1 -10078.075,E2 -10078.075} C_VEL
LIN {X 0,Y 418.671,Z 348.961,A -85,B 0,C 180,E1 -10080,E2 -10080} C_VEL
LIN {X 0,Y 418.509,Z 348.979,A -85,B 0,C 180,E1 -10082.888,E2 -10082.888} C_VEL
LIN {X 0,Y 418.492,Z 348.982,A -85,B 0,C 180,E1 -10086.751,E2 -10086.751} C_VEL
LIN {X 0,Y 418.34,Z 349,A -85,B 0,C 180,E1 -10089.671,E2 -10089.671} C_VEL
LIN {X 0,Y 418.344,Z 348.997,A -85,B 0,C 180,E1 -10093.001,E2 -10093.001} C_VEL
LIN {X 0,Y 418.31,Z 349.004,A -85,B 0,C 180,E1 -10096.736,E2 -10096.736} C_VEL
LIN {X 0,Y 418.269,Z 349.011,A -85,B 0,C 180,E1 -10099.791,E2 -10099.791} C_VEL
LIN {X 0,Y 418.236,Z 349.014,A -85,B 0,C 180,E1 -10102.736,E2 -10102.736} C_VEL
LIN {X 0,Y 418.268,Z 349.012,A -85,B 0,C 180,E1 -10105.904,E2 -10105.904} C_VEL
LIN {X 0,Y 418.272,Z 349.012,A -85,B 0,C 180,E1 -10109.161,E2 -10109.161} C_VEL
LIN {X 0,Y 418.258,Z 349.011,A -85,B 0,C 180,E1 -10112.845,E2 -10112.845} C_VEL
LIN {X 0,Y 418.246,Z 349.014,A -85,B 0,C 180,E1 -10116.239,E2 -10116.239} C_VEL
LIN {X 0,Y 418.253,Z 349.013,A -85,B 0,C 180,E1 -10119.682,E2 -10119.682} C_VEL
LIN {X 0,Y 418.364,Z 349.53,A -85,B 0,C 180,E1 -10120.297,E2 -10120.297} C_VEL
LIN {X 0,Y 419.253,Z 354.822,A -85,B 0,C 180,E1 -10123.879,E2 -10123.879} C_VEL
LIN {X 0,Y 419.971,Z 359.292,A -85,B 0,C 180,E1 -10126.677,E2 -10126.677} C_VEL
LIN {X 0,Y 420.243,Z 362.955,A -85,B 0,C 180,E1 -10128.813,E2 -10128.813} C_VEL
LIN {X 0,Y 419.788,Z 368.659,A -85,B 0,C 180,E1 -10131.893,E2 -10131.893} C_VEL
LIN {X 0,Y 419.322,Z 375.168,A -85,B 0,C 180,E1 -10135.261,E2 -10135.261} C_VEL
LIN {X 0,Y 418.862,Z 382.379,A -85,B 0,C 180,E1 -10138.839,E2 -10138.839} C_VEL
LIN {X 0,Y 418.391,Z 388.788,A -85,B 0,C 180,E1 -10141.944,E2 -10141.944} C_VEL
LIN {X 0,Y 418.035,Z 395.549,A -85,B 0,C 180,E1 -10145.209,E2 -10145.209} C_VEL
LIN {X 0,Y 417.991,Z 396.091,A -85,B 0,C 180,E1 -10145.466,E2 -10145.466} C_VEL
LIN {X 0,Y 422.774,Z 414.724,A -85,B 0,C 180,E1 -10146.232,E2 -10146.232} C_VEL
LIN {X 0,Y 425.762,Z 429.974,A -85,B 0,C 180,E1 -10146.999,E2 -10146.999} C_VEL
LIN {X 0,Y 426.557,Z 435.63,A -85,B 0,C 180,E1 -10147.318,E2 -10147.318} C_VEL
LIN {X 0,Y 425.632,Z 449.294,A -85,B 0,C 180,E1 -10148.064,E2 -10148.064} C_VEL
LIN {X 0,Y 424.358,Z 463.23,A -85,B 0,C 180,E1 -10149.014,E2 -10149.014} C_VEL
LIN {X 0,Y 423.143,Z 476.011,A -85,B 0,C 180,E1 -10150.094,E2 -10150.094} C_VEL
LIN {X 0,Y 421.835,Z 488.947,A -85,B 0,C 180,E1 -10151.42,E2 -10151.42} C_VEL
LIN {X 0,Y 420.805,Z 499.791,A -85,B 0,C 180,E1 -10152.756,E2 -10152.756} C_VEL
LIN {X 0,Y 419.69,Z 509.825,A -85,B 0,C 180,E1 -10154.21,E2 -10154.21} C_VEL
LIN {X 0,Y 418.778,Z 519.656,A -85,B 0,C 180,E1 -10155.917,E2 -10155.917} C_VEL
LIN {X 0,Y 418.164,Z 527.872,A -85,B 0,C 180,E1 -10157.627,E2 -10157.627} C_VEL
LIN {X 0,Y 417.665,Z 534.665,A -85,B 0,C 180,E1 -10159.334,E2 -10159.334} C_VEL
LIN {X 0,Y 417.301,Z 540.947,A -85,B 0,C 180,E1 -10161.282,E2 -10161.282} C_VEL
LIN {X 0,Y 417.152,Z 545.812,A -85,B 0,C 180,E1 -10163.228,E2 -10163.228} C_VEL
LIN {X 0,Y 417.081,Z 549.379,A -85,B 0,C 180,E1 -10165.167,E2 -10165.167} C_VEL
LIN {X 0,Y 417.071,Z 551.727,A -85,B 0,C 180,E1 -10167.103,E2 -10167.103} C_VEL
LIN {X 0,Y 417.052,Z 552.907,A -85,B 0,C 180,E1 -10169.035,E2 -10169.035} C_VEL
LIN {X 0,Y 417.052,Z 552.906,A -85,B 0,C 180,E1 -10170.966,E2 -10170.966} C_VEL
LIN {X 0,Y 417.072,Z 551.72,A -85,B 0,C 180,E1 -10172.898,E2 -10172.898} C_VEL
LIN {X 0,Y 417.091,Z 549.37,A -85,B 0,C 180,E1 -10174.833,E2 -10174.833} C_VEL
LIN {X 0,Y 417.165,Z 545.807,A -85,B 0,C 180,E1 -10176.773,E2 -10176.773} C_VEL
LIN {X 0,Y 417.302,Z 540.94,A -85,B 0,C 180,E1 -10178.719,E2 -10178.719} C_VEL
LIN {X 0,Y 417.666,Z 534.648,A -85,B 0,C 180,E1 -10180.667,E2 -10180.667} C_VEL
LIN {X 0,Y 418.205,Z 526.751,A -85,B 0,C 180,E1 -10182.619,E2 -10182.619} C_VEL
LIN {X 0,Y 418.905,Z 518.363,A -85,B 0,C 180,E1 -10184.328,E2 -10184.328} C_VEL
LIN {X 0,Y 419.844,Z 508.268,A -85,B 0,C 180,E1 -10186.034,E2 -10186.034} C_VEL
LIN {X 0,Y 420.961,Z 497.958,A -85,B 0,C 180,E1 -10187.489,E2 -10187.489} C_VEL
LIN {X 0,Y 422.164,Z 485.678,A -85,B 0,C 180,E1 -10188.943,E2 -10188.943} C_VEL
LIN {X 0,Y 423.529,Z 472.022,A -85,B 0,C 180,E1 -10190.268,E2 -10190.268} C_VEL
LIN {X 0,Y 424.81,Z 458.342,A -85,B 0,C 180,E1 -10191.344,E2 -10191.344} C_VEL
LIN {X 0,Y 425.96,Z 444.181,A -85,B 0,C 180,E1 -10192.238,E2 -10192.238} C_VEL
LIN {X 0,Y 426.594,Z 435.257,A -85,B 0,C 180,E1 -10192.694,E2 -10192.694} C_VEL
LIN {X 0,Y 423.954,Z 420.33,A -85,B 0,C 180,E1 -10193.498,E2 -10193.498} C_VEL
LIN {X 0,Y 420.452,Z 405.533,A -85,B 0,C 180,E1 -10194.164,E2 -10194.164} C_VEL
LIN {X 0,Y 417.982,Z 396.084,A -85,B 0,C 180,E1 -10194.531,E2 -10194.531} C_VEL
LIN {X 0,Y 418.35,Z 389.894,A -85,B 0,C 180,E1 -10197.515,E2 -10197.515} C_VEL
LIN {X 0,Y 418.72,Z 384.223,A -85,B 0,C 180,E1 -10200.235,E2 -10200.235} C_VEL
LIN {X 0,Y 419.185,Z 377.417,A -85,B 0,C 180,E1 -10203.592,E2 -10203.592} C_VEL
LIN {X 0,Y 419.652,Z 370.534,A -85,B 0,C 180,E1 -10207.078,E2 -10207.078} C_VEL
LIN {X 0,Y 420.163,Z 363.741,A -85,B 0,C 180,E1 -10210.719,E2 -10210.719} C_VEL
LIN {X 0,Y 420.114,Z 360.451,A -85,B 0,C 180,E1 -10212.603,E2 -10212.603} C_VEL
LIN {X 0,Y 419.481,Z 356.103,A -85,B 0,C 180,E1 -10215.278,E2 -10215.278} C_VEL
LIN {X 0,Y 418.811,Z 352.182,A -85,B 0,C 180,E1 -10217.838,E2 -10217.838} C_VEL
LIN {X 0,Y 418.251,Z 349.013,A -85,B 0,C 180,E1 -10220.162,E2 -10220.162} C_VEL
LIN {X 0,Y 418.248,Z 349.016,A -85,B 0,C 180,E1 -10222.777,E2 -10222.777} C_VEL
LIN {X 0,Y 418.251,Z 349.015,A -85,B 0,C 180,E1 -10226.323,E2 -10226.323} C_VEL
LIN {X 0,Y 418.247,Z 349.013,A -85,B 0,C 180,E1 -10229.728,E2 -10229.728} C_VEL
LIN {X 0,Y 418.307,Z 349.005,A -85,B 0,C 180,E1 -10233.023,E2 -10233.023} C_VEL
LIN {X 0,Y 418.29,Z 349.006,A -85,B 0,C 180,E1 -10236.219,E2 -10236.219} C_VEL
LIN {X 0,Y 418.253,Z 349.011,A -85,B 0,C 180,E1 -10239.337,E2 -10239.337} C_VEL
LIN {X 0,Y 418.291,Z 349.006,A -85,B 0,C 180,E1 -10242.396,E2 -10242.396} C_VEL
LIN {X 0,Y 418.306,Z 349.006,A -85,B 0,C 180,E1 -10245.403,E2 -10245.403} C_VEL
LIN {X 0,Y 418.319,Z 349.004,A -85,B 0,C 180,E1 -10248.369,E2 -10248.369} C_VEL
LIN {X 0,Y 418.517,Z 348.982,A -85,B 0,C 180,E1 -10252.28,E2 -10252.28} C_VEL
LIN {X 0,Y 418.516,Z 348.978,A -85,B 0,C 180,E1 -10254.217,E2 -10254.217} C_VEL
LIN {X 0,Y 418.548,Z 348.975,A -85,B 0,C 180,E1 -10258.076,E2 -10258.076} C_VEL
LIN {X 0,Y 418.674,Z 348.958,A -85,B 0,C 180,E1 -10260,E2 -10260} C_VEL
LIN {X 0,Y 418.513,Z 348.978,A -85,B 0,C 180,E1 -10262.888,E2 -10262.888} C_VEL
LIN {X 0,Y 418.498,Z 348.976,A -85,B 0,C 180,E1 -10266.751,E2 -10266.751} C_VEL
LIN {X 0,Y 418.345,Z 348.998,A -85,B 0,C 180,E1 -10269.671,E2 -10269.671} C_VEL
LIN {X 0,Y 418.35,Z 348.978,A -85,B 0,C 180,E1 -10273.001,E2 -10273.001} C_VEL
LIN {X 0,Y 418.317,Z 349.004,A -85,B 0,C 180,E1 -10276.736,E2 -10276.736} C_VEL
LIN {X 0,Y 418.274,Z 348.992,A -85,B 0,C 180,E1 -10279.79,E2 -10279.79} C_VEL
LIN {X 0,Y 418.235,Z 349.011,A -85,B 0,C 180,E1 -10282.736,E2 -10282.736} C_VEL
LIN {X 0,Y 418.271,Z 349.001,A -85,B 0,C 180,E1 -10285.904,E2 -10285.904} C_VEL
LIN {X 0,Y 418.268,Z 349.008,A -85,B 0,C 180,E1 -10289.162,E2 -10289.162} C_VEL
LIN {X 0,Y 418.261,Z 349.003,A -85,B 0,C 180,E1 -10292.844,E2 -10292.844} C_VEL
LIN {X 0,Y 418.252,Z 349.013,A -85,B 0,C 180,E1 -10296.239,E2 -10296.239} C_VEL
LIN {X 0,Y 418.258,Z 349.012,A -85,B 0,C 180,E1 -10299.681,E2 -10299.681} C_VEL
LIN {X 0,Y 418.233,Z 349.017,A -85,B 0,C 180,E1 -10302.321,E2 -10302.321} C_VEL
LIN {X 0,Y 418.242,Z 349.015,A -85,B 0,C 180,E1 -10305.109,E2 -10305.109} C_VEL
LIN {X 0,Y 418.179,Z 349.023,A -85,B 0,C 180,E1 -10307.759,E2 -10307.759} C_VEL
LIN {X 0,Y 417.96,Z 349.05,A -85,B 0,C 180,E1 -10310.669,E2 -10310.669} C_VEL
LIN {X 0,Y 417.865,Z 349.063,A -85,B 0,C 180,E1 -10311.516,E2 -10311.516} C_VEL
LIN {X 0,Y 417.792,Z 351.818,A -85,B 0,C 180,E1 -10315.114,E2 -10315.114} C_VEL
LIN {X 0,Y 417.674,Z 354.682,A -85,B 0,C 180,E1 -10318.558,E2 -10318.558} C_VEL
LIN {X 0,Y 417.579,Z 357.612,A -85,B 0,C 180,E1 -10321.884,E2 -10321.884} C_VEL
LIN {X 0,Y 417.547,Z 361.213,A -85,B 0,C 180,E1 -10325.551,E2 -10325.551} C_VEL
LIN {X 0,Y 422.831,Z 376.427,A -85,B 0,C 180,E1 -10326.273,E2 -10326.273} C_VEL
LIN {X 0,Y 427.216,Z 391.01,A -85,B 0,C 180,E1 -10327.108,E2 -10327.108} C_VEL
LIN {X 0,Y 427.521,Z 393.746,A -85,B 0,C 180,E1 -10327.261,E2 -10327.261} C_VEL
LIN {X 0,Y 426.651,Z 407.779,A -85,B 0,C 180,E1 -10327.991,E2 -10327.991} C_VEL
LIN {X 0,Y 425.678,Z 420.561,A -85,B 0,C 180,E1 -10328.828,E2 -10328.828} C_VEL
LIN {X 0,Y 424.469,Z 433.887,A -85,B 0,C 180,E1 -10329.906,E2 -10329.906} C_VEL
LIN {X 0,Y 423.18,Z 446.888,A -85,B 0,C 180,E1 -10331.197,E2 -10331.197} C_VEL
LIN {X 0,Y 421.992,Z 458.225,A -85,B 0,C 180,E1 -10332.555,E2 -10332.555} C_VEL
LIN {X 0,Y 420.898,Z 468.367,A -85,B 0,C 180,E1 -10334.007,E2 -10334.007} C_VEL
LIN {X 0,Y 419.839,Z 478.418,A -85,B 0,C 180,E1 -10335.73,E2 -10335.73} C_VEL
LIN {X 0,Y 419.102,Z 486.499,A -85,B 0,C 180,E1 -10337.408,E2 -10337.408} C_VEL
LIN {X 0,Y 418.295,Z 494.217,A -85,B 0,C 180,E1 -10339.349,E2 -10339.349} C_VEL
LIN {X 0,Y 417.808,Z 500.351,A -85,B 0,C 180,E1 -10341.292,E2 -10341.292} C_VEL
LIN {X 0,Y 417.417,Z 505.457,A -85,B 0,C 180,E1 -10343.403,E2 -10343.403} C_VEL
LIN {X 0,Y 417.21,Z 508.557,A -85,B 0,C 180,E1 -10345.168,E2 -10345.168} C_VEL
LIN {X 0,Y 417.224,Z 510.844,A -85,B 0,C 180,E1 -10347.103,E2 -10347.103} C_VEL
LIN {X 0,Y 417.073,Z 512.037,A -85,B 0,C 180,E1 -10349.137,E2 -10349.137} C_VEL
LIN {X 0,Y 417.082,Z 512.036,A -85,B 0,C 180,E1 -10350.965,E2 -10350.965} C_VEL
LIN {X 0,Y 417.224,Z 510.924,A -85,B 0,C 180,E1 -10352.896,E2 -10352.896} C_VEL
LIN {X 0,Y 417.204,Z 510.48,A -85,B 0,C 180,E1 -10353.339,E2 -10353.339} C_VEL
LIN {X 0,Y 416.545,Z 509.691,A -85,B 0,C 180,E1 -10354.138,E2 -10354.138} C_VEL
LIN {X 0,Y 413.756,Z 508.051,A -85,B 0,C 180,E1 -10355.433,E2 -10355.433} C_VEL
LIN {X 0,Y 411.452,Z 506.395,A -85,B 0,C 180,E1 -10356.468,E2 -10356.468} C_VEL
LIN {X 0,Y 410.534,Z 504.845,A -85,B 0,C 180,E1 -10357.257,E2 -10357.257} C_VEL
LIN {X 0,Y 410.497,Z 504.262,A -85,B 0,C 180,E1 -10357.521,E2 -10357.521} C_VEL
LIN {X 0,Y 410.876,Z 499.565,A -85,B 0,C 180,E1 -10359.351,E2 -10359.351} C_VEL
LIN {X 0,Y 411.404,Z 493.131,A -85,B 0,C 180,E1 -10361.329,E2 -10361.329} C_VEL
LIN {X 0,Y 412.174,Z 486.25,A -85,B 0,C 180,E1 -10363.04,E2 -10363.04} C_VEL
LIN {X 0,Y 412.881,Z 479.139,A -85,B 0,C 180,E1 -10364.541,E2 -10364.541} C_VEL
LIN {X 0,Y 413.987,Z 469.322,A -85,B 0,C 180,E1 -10366.266,E2 -10366.266} C_VEL
LIN {X 0,Y 415.094,Z 459.249,A -85,B 0,C 180,E1 -10367.743,E2 -10367.743} C_VEL
LIN {X 0,Y 416.435,Z 447.624,A -85,B 0,C 180,E1 -10369.167,E2 -10369.167} C_VEL
LIN {X 0,Y 417.725,Z 435.197,A -85,B 0,C 180,E1 -10370.432,E2 -10370.432} C_VEL
LIN {X 0,Y 418.923,Z 422.101,A -85,B 0,C 180,E1 -10371.529,E2 -10371.529} C_VEL
LIN {X 0,Y 419.998,Z 409.613,A -85,B 0,C 180,E1 -10372.376,E2 -10372.376} C_VEL
LIN {X 0,Y 420.942,Z 394.674,A -85,B 0,C 180,E1 -10373.182,E2 -10373.182} C_VEL
LIN {X 0,Y 419.351,Z 388.005,A -85,B 0,C 180,E1 -10373.592,E2 -10373.592} C_VEL
LIN {X 0,Y 414.866,Z 373.825,A -85,B 0,C 180,E1 -10374.401,E2 -10374.401} C_VEL
LIN {X 0,Y 410.48,Z 361.726,A -85,B 0,C 180,E1 -10374.994,E2 -10374.994} C_VEL
LIN {X 0,Y 410.451,Z 361.349,A -85,B 0,C 180,E1 -10375.041,E2 -10375.041} C_VEL
LIN {X 0,Y 410.536,Z 358.047,A -85,B 0,C 180,E1 -10378.641,E2 -10378.641} C_VEL
LIN {X 0,Y 410.645,Z 355.097,A -85,B 0,C 180,E1 -10382.042,E2 -10382.042} C_VEL
LIN {X 0,Y 410.735,Z 352.178,A -85,B 0,C 180,E1 -10385.574,E2 -10385.574} C_VEL
LIN {X 0,Y 410.819,Z 350.192,A -85,B 0,C 180,E1 -10388.1,E2 -10388.1} C_VEL
LIN {X 0,Y 411.031,Z 349.91,A -85,B 0,C 180,E1 -10390.521,E2 -10390.521} C_VEL
LIN {X 0,Y 411.158,Z 349.894,A -85,B 0,C 180,E1 -10393.135,E2 -10393.135} C_VEL
LIN {X 0,Y 411.167,Z 349.895,A -85,B 0,C 180,E1 -10395.88,E2 -10395.88} C_VEL
LIN {X 0,Y 411.163,Z 349.895,A -85,B 0,C 180,E1 -10398.771,E2 -10398.771} C_VEL
LIN {X 0,Y 411.21,Z 349.888,A -85,B 0,C 180,E1 -10401.83,E2 -10401.83} C_VEL
LIN {X 0,Y 411.21,Z 349.888,A -85,B 0,C 180,E1 -10405.121,E2 -10405.121} C_VEL
LIN {X 0,Y 411.167,Z 349.887,A -85,B 0,C 180,E1 -10408.003,E2 -10408.003} C_VEL
LIN {X 0,Y 411.222,Z 349.881,A -85,B 0,C 180,E1 -10411.41,E2 -10411.41} C_VEL
LIN {X 0,Y 411.235,Z 349.884,A -85,B 0,C 180,E1 -10414.707,E2 -10414.707} C_VEL
LIN {X 0,Y 411.204,Z 349.882,A -85,B 0,C 180,E1 -10417.913,E2 -10417.913} C_VEL
LIN {X 0,Y 411.223,Z 349.88,A -85,B 0,C 180,E1 -10421.051,E2 -10421.051} C_VEL
LIN {X 0,Y 411.253,Z 349.88,A -85,B 0,C 180,E1 -10424.132,E2 -10424.132} C_VEL
LIN {X 0,Y 411.313,Z 349.859,A -85,B 0,C 180,E1 -10427.166,E2 -10427.166} C_VEL
LIN {X 0,Y 411.306,Z 349.876,A -85,B 0,C 180,E1 -10430.161,E2 -10430.161} C_VEL
LIN {X 0,Y 411.459,Z 349.857,A -85,B 0,C 180,E1 -10433.133,E2 -10433.133} C_VEL
